ACTION Step_A_01_MoveToXY:
CASE StepA.step OF
	100:
		IF moveCmd_X < Ax_P_Limite AND moveCmd_X > Ax_N_Limite THEN
			StepA.step := StepA.step + 1;
		ELSIF moveCmd_X >= Ax_P_Limite THEN
			StepA.step := StepA.step + 10000;
			pMsg.Push_Alarm("GroupA MoveXY:命令位置超出X軸+極限");
		ELSE
			StepA.step := StepA.step + 10000;
			pMsg.Push_Alarm("GroupA MoveXY:命令位置超出X軸-極限");
		END_IF
 
			
	101:
		IF moveCmd_Y < Ay_P_Limite AND moveCmd_Y > Ay_N_Limite THEN
			StepA.step := StepA.step + 1;
		ELSIF moveCmd_Y >= Ay_P_Limite THEN
			StepA.step := StepA.step + 10000;
			pMsg.Push_Alarm("GroupA MoveXY:命令位置超出Y軸+極限");
		ELSE
			StepA.step := StepA.step + 10000;
			pMsg.Push_Alarm("GroupA MoveXY:命令位置超出Y軸-極限");
		END_IF
		
	102:
		StepA.step := 110;
		
	110:
		Ax.AbsMove(moveCmd_X, moveCmd_Spd);
		Ay.AbsMove(moveCmd_Y, moveCmd_Spd);
		StepA.step := StepA.step + 1;
		
	111:
		IF (Axs.bBuzy OR Axs.bError) AND (Ays.bBuzy OR Ays.bError) THEN
			StepA.step := StepA.step + 1;
		END_IF
		
	112:
		IF Axs.bDone AND Ays.bDone THEN
			StepA.step := StepA.step + 1;
		ELSIF Axs.bError OR Ays.bError THEN
			StepA.step := StepA.step + 10000;
		END_IF
		
	113:
		StepA.bDone := TRUE;
		StepA.step := 0;
		
END_CASE
END_ACTION

ACTION Step_A_02_FindZ:
CASE StepA.step OF
	200:
		IF ProjectData.Now_Steel.Height <= 200 OR 
			Ay.Pos > posc.pos_GbY_stanby THEN
			
			StepA.step := 210;
		ELSE
			StepA.step := 213;
		END_IF
		
		
	210:
		Ax.AbsMove(posc.pos_GbX_stanby, SpdC.HighSpeed);
		Ay.AbsMove(posc.pos_GbY_stanby, SpdC.HighSpeed);
		StepA.step := StepA.step + 1;
		
	211:
		IF (Axs.bBuzy OR Azs.bError) AND (Ays.bBuzy OR Ays.bError) THEN
			StepA.step := StepA.step + 1;
		END_IF
		
	212:
		IF Axs.bDone AND Ays.bDone THEN
			StepA.step := StepA.step + 1;
		ELSIF Axs.bError OR Ays.bError THEN
			StepA.step := StepA.step + 10000;
		END_IF
		
		
	213:
		tmpPos_Z := (ProjectData.Now_Steel.Width / 2) + MaCfg.laserB_Dis + MaCfg.laserB_Z_ReferencePos;
		Az.AbsMove(tmpPos_Z, SpdC.HighSpeed);
		StepA.step := StepA.step + 1;
		
	214:
		IF Azs.bBuzy OR Azs.bError THEN
			StepA.step := StepA.step + 1;
		END_IF
		
	215:
		IF Azs.bDone THEN
			StepA.step := StepA.step + 1;
		ELSIF DisSensor_Dis > 0 AND DisSensor_Dis < 50 THEN
			 Az.Stop();
			 StepA.step := StepA.step + 1;
		ELSIF Azs.bError THEN
			StepA.step := StepA.step + 10000;
		END_IF
		
	216:
		tmr01A.IN := TRUE;
		tmr01A.PT := T#2S;
		IF tmr01A.Q THEN
			tmr01A.IN := FALSE;
			StepA.step := StepA.step + 1;
		END_IF
		
	217:
		StepA.step := 220;
		
		
	220:
		tmpPos_X := macfg.laserB_X_DisSensor2LaserCenter + 10;
		IF ProjectData.Now_Steel.Height > 200 THEN
			tmpPos_Y := (macfg.laserB_Y_ReferencePos - ProjectData.Now_Steel.Height) + 150;
		ELSE
			tmpPos_Y := (macfg.laserB_Y_ReferencePos - MaCfg.laserB_Y_DisSensor2LaserCenter) - 50;
		END_IF
		
		StepA.step := StepA.step + 1;
		
	221:
		Ax.AbsMove(tmpPos_X, SpdC.HighSpeed);
		Ay.AbsMove(tmpPos_Y, SpdC.HighSpeed);
		StepA.step := StepA.step + 1;
		
	222:
		IF (Axs.bBuzy OR Axs.bError) AND (Ays.bBuzy OR Ays.bError) THEN
			StepA.step := StepA.step + 1;
		END_IF
		
	223:
		IF Axs.bDone AND Ays.bDone THEN
			StepA.step := StepA.step + 1;
		ELSIF Axs.bError OR Ays.bError THEN
			StepA.step := StepA.step + 10000;
		END_IF
		
	224:
		StepA.step := 230;
		
		
	230: // 再280-310之間
		IF 280 < DisSensor_Dis AND DisSensor_Dis < 310 THEN
			StepA.step := 240;
		ELSE
			StepA.step := StepA.step + 1;
		END_IF
		
	231:
		Ay.AbsMove(_Position:= PosC.GbX_P_Limite - 120, SpdC.DotSpeed);
		StepA.step := StepA.step + 1;
		
	232:
		IF (280 < DisSensor_Dis AND DisSensor_Dis < 310) OR Ays.bBuzy OR Ays.bError THEN
			StepA.step := StepA.step + 1;
		END_IF
		
	233:
		IF (280 < DisSensor_Dis AND DisSensor_Dis < 310) THEN
			Ay.Stop();
			StepA.step := StepA.step + 1;
		ELSIF Ays.bDone THEN
			pMsg.Push_Error("GroupB_FindZ:再有效距離內找不到可量測的點");
			StepA.step := StepA.step + 10000;
		ELSIF Ays.bError THEN
			StepA.step := StepA.step + 10000;
		END_IF
		
	234:
		tmr01A.IN := TRUE;
		tmr01A.PT := T#2S;
		IF tmr01A.Q THEN
			tmr01A.IN := FALSE;
			StepA.step := StepA.step + 1;
		END_IF
		
	235:
		Ay.RelMove(3, SpdC.LowSpeed);
		StepA.step := StepA.step + 1;
		
	236:
		IF Ays.bBuzy OR Ays.bError THEN
			StepA.step := StepA.step + 1;
		END_IF
		
	237:
		IF Ays.bDone THEN
			StepA.step := StepA.step + 1;
		ELSIF Ays.bError THEN
			StepA.step := StepA.step + 10000;
		END_IF
		
	238:
		StepA.step := 240;
		
		
	240:
		moveZdis := DisSensor_Dis - Macfg.laserB_Dis;
		StepA.step := StepA.step + 1;
	
	241:
		Az.RelMove(moveZdis * -1, SpdC.HighSpeed);
		StepA.step := StepA.step + 1;
		
	242:
		IF Azs.bBuzy OR Azs.bError THEN
			StepA.step := StepA.step + 1;
		END_IF
		
	243:
		IF Azs.bDone THEN
			StepA.step := StepA.step + 1;
		ELSIF Azs.bError THEN
			StepA.step := StepA.step + 10000;
		END_IF
		
	244:
		tmr01A.IN := TRUE;
		tmr01A.PT := T#2S;
		IF tmr01A.Q THEN
			tmr01A.IN := FALSE;
			StepA.step := StepA.step + 1;
		END_IF
		
	245:
		StepA.step := 250;
		
		
	250:
		moveZdis := DisSensor_Dis - Macfg.laserB_Dis;
		IF ProjectData.Now_Steel.Height > 200 THEN
			tmpPos_Y := (macfg.laserB_Y_ReferencePos - ProjectData.Now_Steel.Height) + 125;
		ELSE
			tmpPos_Y := macfg.laserB_Y_ReferencePos - (ProjectData.Now_Steel.Height / 2);
		END_IF
		StepA.step := StepA.step + 1;
		
	251:
		Az.RelMove(moveZdis * -1, SpdC.LowSpeed);
		Ay.AbsMove(tmpPos_Y, SpdC.HighSpeed);
		StepA.step := StepA.step + 1;
		
	252:
		IF (Ays.bBuzy OR Ays.bError) AND (Azs.bBuzy OR Azs.bError) THEN
			StepA.step := StepA.step + 1;
		END_IF
		
	253:
		IF Ays.bDone AND Azs.bDone THEN
			StepA.step := StepA.step + 1;
		ELSIF Azs.bError THEN
			StepA.step := StepA.step + 10000;
		END_IF
		
	254:
		StepA.step := 260;
		
	260:
		z_PosMeasure := Az.Pos;
		StepA.bDone := TRUE;
		StepA.step	:= 0;
		
END_CASE
END_ACTION

ACTION Step_A_03_FindY:
CASE StepA.step OF
	300: // 判斷當距離再200~400間，才做偵測
		IF DisSensor_Dis > 200 OR DisSensor_Dis < 400 THEN
			StepA.step := StepA.step + 1;
		ELSE
			pmsg.Push_Alarm_NoPause("GroupB:Z軸距離感應器不再感應範圍內，取消Y軸原點偵測，使用預設值");
			StepA.step	:= 380;
		END_IF
		
	301:
		StepA.step := 310;
		
	310: 
		Ay.AbsMove(100, 50);
		StepA.step := StepA.step + 1;
		
	311:
		IF Ays.bBuzy OR Ays.bError THEN
			StepA.step := StepA.step + 1;
		END_IF
		
	312:
		IF NOT DisSensor_SSC1 THEN
			Ay.Stop();
			StepA.step := StepA.step + 1;
		ELSIF Ays.bDone THEN
			pmsg.Push_Alarm_NoPause("GroupB:Z軸距離感應器訊號錯誤");
			StepA.step := 380;
		ELSIF Ays.bError THEN
			StepA.step := StepA.step + 10000;
		END_IF
		
	313:
		tmr01A.IN := TRUE;
		tmr01A.PT := T#500MS;
		IF tmr01A.Q THEN
			tmr01A.IN := FALSE;
			StepA.step := StepA.step + 1;
		END_IF
		
	314:
		StepA.step := 320;
		
	320:
		Ay.AbsMove(Ay_P_Limite - 5, 5);
		StepA.step := StepA.step + 1;
		
	321:
		IF (Ays.bBuzy OR Ays.bError) THEN
			StepA.step := StepA.step + 1;
		END_IF
		
	322:
		IF DisSensor_SSC1 THEN
			Ay.Stop();
			StepA.step := StepA.step + 1;
		ELSIF Ays.bDone THEN
			pmsg.Push_Alarm_NoPause("GroupB:Z軸距離感應器訊號錯誤");
			StepA.step := 380;
		ELSIF Ays.bError THEN
			StepA.step := StepA.step + 10000;
		END_IF
		
	323:
		tmr01A.IN := TRUE;
		tmr01A.PT := T#500MS;
		IF tmr01A.Q THEN
			tmr01A.IN := FALSE;
			StepA.step := StepA.step + 1;
		END_IF
		
	324:
		StepA.step := 330;
		
		
	330:
		Ay.AbsMove(100, 0.5);
		StepA.step := StepA.step + 1;
		
	331:
		IF Ays.bBuzy OR Ays.bError THEN
			StepA.step := StepA.step + 1;
		END_IF
		
	332:
		IF NOT DisSensor_SSC1 THEN
			Ay.Stop();
			StepA.step := StepA.step + 1;
		ELSIF Ays.bDone THEN
			pmsg.Push_Alarm_NoPause("GroupB:Z軸距離感應器訊號錯誤");
			StepA.step := 380;
		ELSIF Ays.bError THEN
			StepA.step := StepA.step + 10000;
		END_IF
		
	333:
		tmr01A.IN := TRUE;
		tmr01A.PT := T#500MS;
		IF tmr01A.Q THEN
			tmr01A.IN := FALSE;
			StepA.step := StepA.step + 1;
		END_IF
		
	334:
		StepA.step := 340;
		
		
	340:
		Set_Y_Ref(Ay.Pos);
		StepA.step := StepA.step + 1;
		
	341:
		StepA.step := 390;
		
	
	380:
		IF projectData.Now_Steel.Height > 0 THEN
			Set_Y_Ref(Ay_P_Limite + 56 - projectData.Now_Steel.Height);
		ELSE
			Set_Y_Ref(Ay_P_Limite + 56 - 500);
		END_IF
		StepA.step := StepA.step + 1;
		
	381:
		StepA.step	:= 390;
	
	390:
		StepA.bDone := TRUE;
		StepA.step	:= 0;
		
END_CASE
END_ACTION

ACTION Step_A_10_MoveToXY_REF:
CASE StepA.step OF
	1000:// 計算相對距離
		tmpPos_X := moveCmd_X - pointRef.X;
		tmpPos_Y := moveCmd_Y + pointRef.Y;
		Dxf_Y_Move := 0;
		StepA.step := StepA.step + 1;
		
	1001:
		IF tmpPos_X < Ax_P_Limite AND tmpPos_X > Ax_N_Limite THEN
			StepA.step := StepA.step + 1;
		ELSIF tmpPos_X >= Ax_P_Limite THEN
			StepA.step := StepA.step + 10000;
			pMsg.Push_Alarm("GroupB MoveXY:命令位置超出X軸+極限");
		ELSE
			StepA.step := StepA.step + 10000;
			pMsg.Push_Alarm("GroupB MoveXY:命令位置超出X軸-極限");
		END_IF
 
			
	1002:
		IF tmpPos_Y < Ay_P_Limite AND tmpPos_Y > Ay_N_Limite THEN
			StepA.step := StepA.step + 1;
		ELSIF tmpPos_Y >= Ay_P_Limite THEN
			StepA.step := StepA.step + 10000;
			pMsg.Push_Alarm("GroupB MoveXY_Ref:命令位置超出Y軸+極限");
		ELSE
			StepA.step := StepA.step + 10000;
			pMsg.Push_Alarm("GroupB MoveXY_Ref:命令位置超出Y軸-極限");
		END_IF
		
	1003:
		StepA.step := 1010;
		
	1010:
		Ax.AbsMove(tmpPos_X, moveCmd_Spd);
		Ay.AbsMove(tmpPos_Y, moveCmd_Spd);
		StepA.step := StepA.step + 1;
		
	1011:
		IF (Axs.bBuzy OR Axs.bError) AND (Ays.bBuzy OR Ays.bError) THEN
			StepA.step := StepA.step + 1;
		END_IF
		
	1012:
		IF Axs.bDone AND Ays.bDone THEN
			StepA.step := StepA.step + 1;
		ELSIF Axs.bError OR Ays.bError THEN
			StepA.step := StepA.step + 10000;
		END_IF
		
	1013:
		tmr01A.IN := TRUE;
		tmr01A.PT := T#1S;
		IF tmr01A.Q THEN
			tmr01A.IN := FALSE;
			StepA.step := StepA.step + 1;
		END_IF
		
	1014:
		StepA.step := 1020;
		
	1020:
		StepA.bDone := TRUE;
		StepA.step := 0;
		
END_CASE
END_ACTION

ACTION Step_A_20_ToStanbyPos:
CASE StepA.step OF
	2000:
		StepA.step := 2010;
		
	2010:
		IF Az.Pos > posc.pos_GbZ_stanby - 20 THEN
			StepA.step := 2020;
		ELSE
			StepA.step := StepA.step + 1;
		END_IF
		
	2011:
		Az.RelMove(20, SpdC.HomeSpeed);
		StepA.step := StepA.step + 1;
		
	2012:
		IF Azs.bDone OR Azs.bError OR NOT GbZ.outLimiter THEN
			StepA.step := StepA.step + 1;
		END_IF
		
	2013:
		IF Azs.bDone OR NOT GbZ.outLimiter THEN
			StepA.step := StepA.step + 1;
		ELSIF Azs.bError THEN
			StepA.step := StepA.step + 10000;
		END_IF
		
	2014:
		StepA.step := 2020;
		
	2020:
		Ax.AbsMove(posc.pos_GbX_stanby, moveCmd_Spd);
		StepA.step := StepA.step + 1;
		
	2021:
		IF (Axs.bBuzy OR Axs.bError) THEN
			StepA.step := StepA.step + 1;
		END_IF
		
	2022:
		IF Axs.bDone THEN
			StepA.step := StepA.step + 1;
		ELSIF Axs.bError THEN
			StepA.step := StepA.step + 10000;
		END_IF
	
	2023:
		StepA.step := 2030;
	
	2030:
		Az.AbsMove(posc.pos_GbZ_stanby, moveCmd_Spd);
		Ay.AbsMove(posc.pos_GbY_stanby, moveCmd_Spd);
		StepA.step := StepA.step + 1;
		
	2031:
		IF (Azs.bBuzy OR Azs.bError) AND (Ays.bBuzy OR Ays.bError)  THEN
			StepA.step := StepA.step + 1;
		END_IF
		
	2032:
		IF Azs.bDone AND Ays.bDone THEN
			StepA.step := StepA.step + 1;
		ELSIF Azs.bError OR Ays.bError THEN
			StepA.step := StepA.step + 10000;
		END_IF
		
	2033:
		StepA.step := 2040;
		
		
	2040:
		StepA.bDone := TRUE;
		StepA.step := 0;
		
END_CASE
END_ACTION

ACTION Timer:
tmr01A();
tmr01();
tmr02();

// tmr_oil(in := IO.q205 AND IO.i402, PT:=T#2S);
tmr_oil(in := IO.q205, PT:=T#2S);

IF tmr_oil.Q THEN
	IO.q205 := FALSE;
	
	Axis.GbX_Last_Oil := Axis.GbX_total_Move;
	
	Axis.GbY_Last_Oil := Axis.GbY_total_Move;
	
	Axis.GbZ_Last_Oil := Axis.GbZ_total_Move;
END_IF
END_ACTION

METHOD ToStanby : BOOL
VAR_INPUT
	Speed : LREAL := 0;
END_VAR
StepA.bDone := FALSE;
IF Speed > 0 THEN
	moveCmd_Spd := Speed;
ELSE
	moveCmd_Spd := SpdC.HomeSpeed;
END_IF

// ============ 紀錄啟動條件 ============
_logA.fbJson.StartObject();
_logA.fbJson.AddKeyString('MethodName','ToStanby');
_logA.fbJson.AddKeyLreal('Velocity', Speed);
_logA.JsonOutput();
// ======================================



StepA.step := 2000;
END_METHOD

METHOD XY_Move : BOOL
VAR_INPUT
	X_Point : REAL;
	Y_Point	: REAL;
	Speed : REAL;
END_VAR
moveCmd_X := X_Point;
moveCmd_Y := Y_Point;
moveCmd_Spd := Speed;

StepA.bDone := FALSE;

// ============ 紀錄啟動條件 ============
_logA.fbJson.StartObject();
_logA.fbJson.AddKeyString('MethodName','XY_Move');
_logA.fbJson.AddKeyLreal('X_Point', X_Point);
_logA.fbJson.AddKeyLreal('Y_Point', Y_Point);
_logA.fbJson.AddKeyLreal('Velocity', Speed);
_logA.JsonOutput();
// ======================================



StepA.step := 100;
END_METHOD

METHOD XY_Move_Ref : BOOL
VAR_INPUT
	X_Point : LREAL;
	Y_Point	: LREAL;
	Speed : LREAL;
END_VAR
moveCmd_X := X_Point;
moveCmd_Y := Y_Point;
moveCmd_Spd := Speed;

StepA.bDone := FALSE;

// ============ 紀錄啟動條件 ============
_logA.fbJson.StartObject();
_logA.fbJson.AddKeyString('MethodName','XY_Move_Ref');
_logA.fbJson.AddKeyLreal('X_Point', X_Point);
_logA.fbJson.AddKeyLreal('Y_Point', Y_Point);
_logA.fbJson.AddKeyLreal('Velocity', Speed);
_logA.JsonOutput();
// ======================================



StepA.step := 1000;
END_METHOD

END_PROGRAM

// ---- POUs/動作流程控制/AxisGroup功能塊/GroupC.TcPOU
PROGRAM GroupC
VAR
	step		: INT;
	
	StepA		: Sub_Step;
	
	// X軸映射
	Ax : I_Axis;
	Axs: Sub_Step;
	// Y軸映射
	Ay : I_Axis;
	Ays: Sub_Step;
	// X軸映射
	Az : I_Axis;
	Azs: Sub_Step;
	
	Ax_P_Limite : LREAL;
	Ax_N_Limite : LREAL;
	Ay_P_Limite : LREAL;
	Ay_N_Limite : LREAL;
	Az_P_Limite : LREAL;
	Az_N_Limite : LREAL;

	
	// 移動命令的 X位置
	moveCmd_X: LREAL;
	// 移動命令的 Y位置
	moveCmd_Y: LREAL;
	// 移動命令 速度
	moveCmd_Spd: LREAL;
	
	moveZdis	: REAL;
	tmr01A		: TON;
	tmr01		: TON;
	tmr02		: TON;
	
	// 坐標系的參考原點
	pointRef : XYZ_Point;
	
	// 移動位置X 計算結果
	tmpPos_X: LREAL;
	// 移動位置Y 計算結果
	tmpPos_Y: LREAL;
	// 移動位置Z 計算結果
	tmpPos_Z: LREAL;
	
	// 雷射圖形移動距離 Y
	Dxf_Y_Move : LREAL;
	

	// 測量到的Z位置
	z_PosMeasure: REAL;
	
	// 距離感應器IO
	DisSensor_SSC1: BOOL;
	// 距離感應器距離
	DisSensor_Dis: LREAL;
	
	Boot : BOOL := TRUE;
	
	
	
	// 執行中的清單號
	WorkNum: INT;
	
	// 鏡頭 吹氣
	q_Lens_Blow :BOOL;
	
	// 重試計數器
	_retryCnt: INT;
	
	// 可以開始雕刻 (Fx就緒)
	_ReadyToPrint :BOOL;
	// 可以開始移動 (Fx就緒)
	_ReadyToMove :BOOL;
	
	
	// 計算上次打油後的一棟距離
	X_Move: LREAL;
	Y_Move: LREAL;
	Z_Move: LREAL;
	tmr_oil: TON;
	
	_log : Step_Log; 
	_logA : Step_Log; 
	sql_hand: UDINT;
END_VAR



VAR_OUTPUT
	// 工件高度
	Size_H : REAL;
	// 工件座標
	RefPos : XYZ_Point;
	
	// 功能執行中
	bBuzy 	: BOOL;
	// 功能結束
	bDone	: BOOL;
	// 發生錯誤
	bError	: BOOL;
END_VAR

IF Boot THEN
	Ax := axis.GcX;
	Ay := axis.GcY;
	Az := axis.GcZ;
	boot := FALSE;
END_IF

Axs := Ax.State;
Ays := Ay.State;
Azs := Az.State;

Ax_P_Limite := posc.GcX_P_Limite;
Ax_N_Limite := posc.GcX_N_Limite;
Ay_P_Limite := posc.GcY_P_Limite;
Ay_N_Limite := posc.GcY_N_Limite;
Az_P_Limite := posc.GcZ_P_Limite;
Az_N_Limite := posc.GcZ_N_Limite;

DisSensor_SSC1	:= Sensor.sensorC.SSC1_1;
DisSensor_Dis	:= Sensor.sensorC.Distance;

IF (EStop OR SystemError) THEN
	IF bBuzy THEN
		step := step  + 10000;
	END_IF
	IF StepA.bBuzy THEN
		StepA.step := StepA.step  + 10000;
	END_IF
	Hmi_Web.Process_Data_UUID_C_Start := FALSE;
	q_Lens_Blow := FALSE;
END_IF

bBuzy := step > 0 AND step < 10000;
bError := step >= 10000;
IF bBuzy OR bError THEN
	bDone := FALSE;
END_IF

Step_01_DoPayloadList();
Step_02_Do_2nd_in_list();
Step_03_DoLaserAction();



StepA.bBuzy := StepA.step > 0 AND StepA.step < 10000;
StepA.bError := StepA.step >= 10000;
IF StepA.bBuzy OR StepA.bError THEN
	StepA.bDone := FALSE;
END_IF

Step_A_01_MoveToXY();
Step_A_02_FindZ();
Step_A_03_FindY();
Step_A_10_MoveToXY_REF();
Step_A_20_ToStanbyPos();

Timer();

RefPos.X := Ax.Pos - pointRef.X;
RefPos.Y := Ay.Pos - pointRef.Y;
RefPos.Z := Az.Pos - pointRef.Z;

ProjectData.Now_Steel_Payload_C_DataNumberDone := WorkNum;

io.q307 := q_Lens_Blow;

_log(name:= 'GroupC', step:= step);
_logA(name:= 'GroupC_Mov', step:= StepA.Step);

METHOD Do_WorkList : BOOL
VAR_INPUT
END_VAR
bDone := FALSE;

// ============ 紀錄啟動條件 ============
_log.fbJson.StartObject();
_log.fbJson.AddKeyString('MethodName','Do_WorkList');
_log.JsonOutput();
// ======================================




Step := 100;
END_METHOD

METHOD FindZ : BOOL
VAR_INPUT
END_VAR
StepA.bDone := FALSE;

// ============ 紀錄啟動條件 ============
_logA.fbJson.StartObject();
_logA.fbJson.AddKeyString('MethodName','FindZ');
_logA.JsonOutput();
// ======================================






StepA.step := 200;
END_METHOD

METHOD FindZ_Fast : BOOL
VAR_INPUT
END_VAR
StepA.bDone := FALSE;

// ============ 紀錄啟動條件 ============
_logA.fbJson.StartObject();
_logA.fbJson.AddKeyString('MethodName','FindZ_Fast');
_logA.JsonOutput();
// ======================================





StepA.step := 220;
END_METHOD

ACTION Oil:
X_Move := Axis.GcX_total_Move - Axis.GcX_Last_Oil;
Y_Move := Axis.GcY_total_Move - Axis.GcY_Last_Oil;
Z_Move := Axis.GcZ_total_Move - Axis.GcZ_Last_Oil;

IF X_Move > 1000000 OR Y_Move > 1000000 OR Z_Move > 1000000 THEN
	IO.q206 := TRUE;
END_IF
END_ACTION

PROPERTY ReadyToMove : BOOL
GET
ReadyToMove := _ReadyToMove;
END_GET
SET
_ReadyToMove := ReadyToMove;
END_SET
END_PROPERTY

PROPERTY ReadyToPrint : BOOL
GET
ReadyToPrint := _ReadyToPrint;
END_GET
SET
_ReadyToPrint := ReadyToPrint;
END_SET
END_PROPERTY

METHOD Set_X_Ref
VAR_INPUT
	Value : LREAL;
END_VAR
pointRef.X := Value;
END_METHOD

METHOD Set_Y_Ref
VAR_INPUT
	Value : LREAL;
END_VAR
pointRef.Y := Value;
END_METHOD

ACTION Step_01_DoPayloadList:
CASE step OF
(*	===============================================
		開始做 Payload_B_Data_buff 清單內的工作
	===============================================*)
	100: // 以數量判斷是否有工作
		WorkNum := 0;
		IF ProjectData.Now_Steel_Payload_C_DataNumber > 0 THEN
			step := step + 1;
		ELSE
			bDone := TRUE;
			Step := 0;
		END_IF
 
			
	101:
		// 初始化工作暫存器
		Hmi_Web.Process_Data_UUID_A_Start := FALSE;
		WorkNum := 0;
		step := 110;
		
(*	===============================================
					設定工作中的專案
	===============================================*)
	110:
		ProjectData.Payload_C_Data_Now := ProjectData.Payload_C_Data_buff[WorkNum];
		Hmi_Web.Process_Data_UUID_A := ProjectData.Payload_C_Data_buff[WorkNum].data_uid;
		step := step + 1;
	
	111:
		step := 120;
		
(*	===============================================
					移動到位置
	===============================================*)
	120:
		IF _ReadyToMove THEN
			step := step + 1;
		END_IF
		
	121:
		XY_Move_Ref(
			ProjectData.Payload_C_Data_Now.Point_X, 
			ProjectData.Payload_C_Data_Now.Point_Y, 
			SpdC.HighSpeed
		);
		step := step + 1;
		
	122:
		IF stepA.bBuzy OR stepA.bError THEN
			step := step + 1;
		END_IF
		
	123:
		IF stepA.bDone THEN
			step := step + 1;
		ELSIF stepA.bError THEN
			step := step + 10000;
		END_IF
		
	124:
		step := 130;
	

(*	===============================================
				雷射主機 啟動 預覽/雕刻 動作
	===============================================*)	
	130:
		step := 300;
END_CASE
END_ACTION

ACTION Step_02_Do_2nd_in_list:
CASE step OF
	200:
		step := 210;
		
(*	===============================================
					設定工作中的專案
	===============================================*)
	210:
		ProjectData.Payload_C_Data_Now := ProjectData.Payload_C_Data_buff[WorkNum];
		Hmi_Web.Process_Data_UUID_A := ProjectData.Payload_C_Data_buff[WorkNum].data_uid;
		step := step + 1;
	
	211:
		step := 220;
		
(*	===============================================
					移動到位置
	===============================================*)
	220:
		XY_Move_Ref(
			ProjectData.Payload_C_Data_Now.Point_X, 
			ProjectData.Payload_C_Data_Now.Point_Y, 
			SpdC.HighSpeed
		);
		step := step + 1;
		
	221:
		IF stepA.bBuzy OR stepA.bError THEN
			step := step + 1;
		END_IF
		
	222:
		IF stepA.bDone THEN
			step := step + 1;
		ELSIF stepA.bError THEN
			step := step + 10000;
		END_IF
		
	223:
		step := 230;

(*	===============================================
				雷射主機 啟動 預覽/雕刻 動作
	===============================================*)	
	230:
		step := 300;
		
END_CASE
END_ACTION

ACTION Step_03_DoLaserAction:
CASE step OF
	300:
		IF ReadyToPrint THEN
			step := step + 1;
		END_IF
		
	301:
		sql_hand := ReadSQLData.Set_Payload_Start(ProjectData.Payload_C_Data_Now.data_uid);
		IF sql_hand <> 0 THEN
			step := step + 1;
		END_IF
		
	302:
		step := 310;

(*	===============================================
				雷射主機 啟動 預覽/雕刻 動作
	===============================================*)	
	310:
		q_Lens_Blow := TRUE;
		IF LEN(Hmi_Web.Process_Data_UUID_A) = 0 THEN
			Hmi_Web.Process_Data_UUID_A := ProjectData.Payload_C_Data_buff[WorkNum].data_uid;
		ELSE
			step := step + 1;
		END_IF
		
	311:
		Hmi_Web.Process_Data_UUID_A_Start := TRUE;
		// ============ 紀錄啟動條件 ============
		_log.fbJson.StartObject();
		_log.fbJson.AddKeyString('StepName','Laser_C_Start');
		_log.fbJson.AddKeyBool('Process_Data_UUID_A_Start', Hmi_Web.Process_Data_UUID_A_Start);
		_log.fbJson.AddKeyString('Payload_C_Data_Now', ProjectData.Payload_C_Data_Now.data_uid);
		_log.JsonOutput();
		// ======================================
		step := step + 1;
		
	312:	
		tmr01.PT := T#500MS;
		tmr01.IN := TRUE;
		IF tmr01.Q THEN
			tmr01.IN := FALSE;
			tmr02.IN := FALSE;
			step := step + 1;
		END_IF
		
	313:
		tmr01.PT := TO_TIME(MaCfg.LaserPrinter_Timeout);
		tmr01.IN := TRUE;
		tmr02.PT := T#250mS;
		tmr02.IN := NOT Hmi_Web.Process_Data_UUID_A_Start;
		IF tmr02.Q THEN
			Hmi_Web.Process_Data_UUID_A :='';
			tmr01.IN := FALSE;
			tmr02.IN := FALSE;
			// ============ 紀錄啟動條件 ============
			_log.fbJson.StartObject();
			_log.fbJson.AddKeyString('StepName','Laser_C_Done');
			_log.JsonOutput();
			// ======================================
			step := step + 1;
		ELSIF tmr01.Q THEN
			tmr01.IN := FALSE;
			tmr02.IN := FALSE;
			pMsg.Push_Error("GroupC:雷射動作超時");
			step := step + 10000;
		END_IF
	
	314:
		WorkNum := WorkNum + 1;
		q_Lens_Blow := FALSE;
		step := 320;
		
(*	================================================
				開始下個循環或此區域結束
	================================================*)	
	320:
		sql_hand := ReadSQLData.Set_Payload_Finish(ProjectData.Payload_C_Data_Now.data_uid);
		IF sql_hand <> 0 THEN
			step := step + 1;
		END_IF
	
	321:
		IF WorkNum < ProjectData.Now_Steel_Payload_C_DataNumber THEN
		// 這個區域還有工作
			step := step + 1;
		ELSE
		// 這個區域工作結束
			step := 390;
		END_IF
		
	322:
		// 設定工作中的專案
		step := 200;
		
(*	================================================
				此區域結束
	================================================*)		
	390:
		bDone := TRUE;
		step := 0;
END_CASE
END_ACTION

ACTION Step_A_01_MoveToXY:
CASE StepA.step OF
	100:
		IF moveCmd_X < Ax_P_Limite AND moveCmd_X > Ax_N_Limite THEN
			StepA.step := StepA.step + 1;
		ELSIF moveCmd_X >= Ax_P_Limite THEN
			StepA.step := StepA.step + 10000;
			pMsg.Push_Alarm("GroupA MoveXY:命令位置超出X軸+極限");
		ELSE
			StepA.step := StepA.step + 10000;
			pMsg.Push_Alarm("GroupA MoveXY:命令位置超出X軸-極限");
		END_IF
 
			
	101:
		IF moveCmd_Y < Ay_P_Limite AND moveCmd_Y > Ay_N_Limite THEN
			StepA.step := StepA.step + 1;
		ELSIF moveCmd_Y >= Ay_P_Limite THEN
			StepA.step := StepA.step + 10000;
			pMsg.Push_Alarm("GroupA MoveXY:命令位置超出Y軸+極限");
		ELSE
			StepA.step := StepA.step + 10000;
			pMsg.Push_Alarm("GroupA MoveXY:命令位置超出Y軸-極限");
		END_IF
		
	102:
		StepA.step := 110;
		
	110:
		Ax.AbsMove(moveCmd_X, moveCmd_Spd);
		Ay.AbsMove(moveCmd_Y, moveCmd_Spd);
		StepA.step := StepA.step + 1;
		
	111:
		IF (Axs.bBuzy OR Axs.bError) AND (Ays.bBuzy OR Ays.bError) THEN
			StepA.step := StepA.step + 1;
		END_IF
		
	112:
		IF Axs.bDone AND Ays.bDone THEN
			StepA.step := StepA.step + 1;
		ELSIF Axs.bError OR Ays.bError THEN
			StepA.step := StepA.step + 10000;
		END_IF
		
	113:
		StepA.bDone := TRUE;
		StepA.step := 0;
		
END_CASE
END_ACTION

ACTION Step_A_02_FindZ:
CASE StepA.step OF
	200:
		StepA.step := 220;
		
	220:
		tmpPos_X := 150;
		tmpPos_Y := (ProjectData.Now_Steel.Width / 2) + pointRef.Y;
		tmpPos_Z := ProjectData.Now_Steel.Height + MaCfg.laserC_Dis + MaCfg.laserC_Z_ReferencePos;
		StepA.step := StepA.step + 1;
		
	221:
		Ax.AbsMove(tmpPos_X, SpdC.HighSpeed);
		Ay.AbsMove(tmpPos_Y, SpdC.HighSpeed);
		Az.AbsMove(tmpPos_Z, SpdC.HighSpeed);
		StepA.step := StepA.step + 1;
		
	222:
		IF (Axs.bBuzy OR Axs.bError) AND 
			(Ays.bBuzy OR Ays.bError) AND
			(Azs.bBuzy OR Azs.bError) THEN
			StepA.step := StepA.step + 1;
		END_IF
		
	223:
		IF Axs.bDone AND Ays.bDone AND Azs.bDone THEN
			StepA.step := StepA.step + 1;
		ELSIF Axs.bError OR Ays.bError OR Azs.bError THEN
			StepA.step := StepA.step + 10000;
		END_IF
		
	224:
		StepA.step := 230;
		
	
	230: // 再280-310之間
		IF 280 < DisSensor_Dis AND DisSensor_Dis < 310 THEN
			StepA.step := 240;
		ELSE
			StepA.step := StepA.step + 1;
		END_IF
		
	231:
		Ay.AbsMove((ProjectData.Now_Steel.Width - 10) + pointRef.Y, SpdC.DotSpeed);
		StepA.step := StepA.step + 1;
		
	232:
		IF (280 < DisSensor_Dis AND DisSensor_Dis < 310) OR Ays.bBuzy OR Ays.bError THEN
			StepA.step := StepA.step + 1;
		END_IF
		
	233:
		IF (280 < DisSensor_Dis AND DisSensor_Dis < 310) THEN
			Ay.Stop();
			StepA.step := StepA.step + 1;
		ELSIF Ays.bDone THEN
			pMsg.Push_Error("GroupC_FindZ:再有效距離內找不到可量測的點");
			StepA.step := StepA.step + 10000;
		ELSIF Ays.bError THEN
			StepA.step := StepA.step + 10000;
		END_IF
		
	234:
		tmr01A.IN := TRUE;
		tmr01A.PT := T#2S;
		IF tmr01A.Q THEN
			tmr01A.IN := FALSE;
			StepA.step := StepA.step + 1;
		END_IF
		
	235:
		Ay.RelMove(3, SpdC.LowSpeed);
		StepA.step := StepA.step + 1;
		
	236:
		IF Ays.bBuzy OR Ays.bError THEN
			StepA.step := StepA.step + 1;
		END_IF
		
	237:
		IF Ays.bDone THEN
			StepA.step := StepA.step + 1;
		ELSIF Ays.bError THEN
			StepA.step := StepA.step + 10000;
		END_IF
		
	238:
		StepA.step := 240;
	
		
	240:
		moveZdis := DisSensor_Dis - Macfg.laserC_Dis;
		StepA.step := StepA.step + 1;
		
		
	241:
		Az.RelMove(moveZdis * -1, SpdC.HighSpeed);
		StepA.step := StepA.step + 1;
		
	242:
		IF Azs.bBuzy OR Azs.bError THEN
			StepA.step := StepA.step + 1;
		END_IF
		
	243:
		IF Azs.bDone THEN
			StepA.step := StepA.step + 1;
		ELSIF Azs.bError THEN
			StepA.step := StepA.step + 10000;
		END_IF
		
	244:
		tmr01A.IN := TRUE;
		tmr01A.PT := T#2S;
		IF tmr01A.Q THEN
			tmr01A.IN := FALSE;
			StepA.step := StepA.step + 1;
		END_IF
		
	245:
		StepA.step := 250;
		
		
	250:
		moveZdis := DisSensor_Dis - Macfg.laserC_Dis;
		StepA.step := StepA.step + 1;
		
	251:
		Az.RelMove(moveZdis * -1, SpdC.LowSpeed);
		StepA.step := StepA.step + 1;
		
	252:
		IF Azs.bBuzy OR Azs.bError THEN
			StepA.step := StepA.step + 1;
		END_IF
		
	253:
		IF Azs.bDone THEN
			StepA.step := StepA.step + 1;
		ELSIF Azs.bError THEN
			StepA.step := StepA.step + 10000;
		END_IF
		
	254:
		StepA.step := 260;
		
	260:
		z_PosMeasure := Az.Pos;
		StepA.bDone := TRUE;
		StepA.step	:= 0;
		
END_CASE
END_ACTION

ACTION Step_A_03_FindY:
CASE StepA.step OF
	300: // 判斷當距離再200~400間，才做偵測
		IF DisSensor_Dis > 200 OR DisSensor_Dis < 400 THEN
			StepA.step := StepA.step + 1;
		ELSE
			pmsg.Push_Alarm_NoPause("GroupC:Z軸距離感應器不再感應範圍內，取消Y軸原點偵測，使用預設值");
			StepA.step	:= 380;
		END_IF
		
	301:
		StepA.step := 310;
		
	310: 
		Ay.AbsMove(100, 50);
		StepA.step := StepA.step + 1;
		
	311:
		IF Ays.bBuzy OR Ays.bError THEN
			StepA.step := StepA.step + 1;
		END_IF
		
	312:
		IF NOT DisSensor_SSC1 THEN
			Ay.Stop();
			StepA.step := StepA.step + 1;
		ELSIF Ays.bDone THEN
			pmsg.Push_Alarm_NoPause("GroupC:Z軸距離感應器訊號錯誤");
			StepA.step := 380;
		ELSIF Ays.bError THEN
			StepA.step := StepA.step + 10000;
		END_IF
		
	313:
		tmr01A.IN := TRUE;
		tmr01A.PT := T#500MS;
		IF tmr01A.Q THEN
			tmr01A.IN := FALSE;
			StepA.step := StepA.step + 1;
		END_IF
		
	314:
		StepA.step := 320;
		
	320:
		Ay.AbsMove(Ay_P_Limite - 5, 5);
		StepA.step := StepA.step + 1;
		
	321:
		IF (Ays.bBuzy OR Ays.bError) THEN
			StepA.step := StepA.step + 1;
		END_IF
		
	322:
		IF DisSensor_SSC1 THEN
			Ay.Stop();
			StepA.step := StepA.step + 1;
		ELSIF Ays.bDone THEN
			pmsg.Push_Alarm_NoPause("GroupC:Z軸距離感應器訊號錯誤");
			StepA.step := 380;
		ELSIF Ays.bError THEN
			StepA.step := StepA.step + 10000;
		END_IF
		
	323:
		tmr01A.IN := TRUE;
		tmr01A.PT := T#500MS;
		IF tmr01A.Q THEN
			tmr01A.IN := FALSE;
			StepA.step := StepA.step + 1;
		END_IF
		
	324:
		StepA.step := 330;
		
		
	330:
		Ay.AbsMove(100, 0.5);
		StepA.step := StepA.step + 1;
		
	331:
		IF Ays.bBuzy OR Ays.bError THEN
			StepA.step := StepA.step + 1;
		END_IF
		
	332:
		IF NOT DisSensor_SSC1 THEN
			Ay.Stop();
			StepA.step := StepA.step + 1;
		ELSIF Ays.bDone THEN
			pmsg.Push_Alarm_NoPause("GroupC:Z軸距離感應器訊號錯誤");
			StepA.step := 380;
		ELSIF Ays.bError THEN
			StepA.step := StepA.step + 10000;
		END_IF
		
	333:
		tmr01A.IN := TRUE;
		tmr01A.PT := T#500MS;
		IF tmr01A.Q THEN
			tmr01A.IN := FALSE;
			StepA.step := StepA.step + 1;
		END_IF
		
	334:
		StepA.step := 340;
		
		
	340:
		Set_Y_Ref(Ay.Pos);
		StepA.step := StepA.step + 1;
		
	341:
		StepA.step := 390;
		
	
	380:
		IF projectData.Now_Steel.Width > 0 THEN
			Set_Y_Ref(Ay_P_Limite + 56 - projectData.Now_Steel.Width);
		ELSE
			Set_Y_Ref(Ay_P_Limite + 56 - 500);
		END_IF
		StepA.step := StepA.step + 1;
		
	381:
		StepA.step	:= 390;
	
	390:
		z_PosMeasure := GaZ.Pos;
		StepA.bDone := TRUE;
		StepA.step	:= 0;
		
END_CASE
END_ACTION

ACTION Step_A_10_MoveToXY_REF:
CASE StepA.step OF
	1000:// 計算相對距離
		tmpPos_X := moveCmd_X - pointRef.X;
		tmpPos_Y := moveCmd_Y + pointRef.Y;
		Dxf_Y_Move := 0;
		StepA.step := StepA.step + 1;
		
	1001:
		IF tmpPos_X < Ax_P_Limite AND tmpPos_X > Ax_N_Limite THEN
			StepA.step := StepA.step + 1;
		ELSIF tmpPos_X >= Ax_P_Limite THEN
			StepA.step := StepA.step + 10000;
			pMsg.Push_Alarm("GroupC MoveXY:命令位置超出X軸+極限");
		ELSE
			StepA.step := StepA.step + 10000;
			pMsg.Push_Alarm("GroupC MoveXY:命令位置超出X軸-極限");
		END_IF
 
			
	1002:
		IF tmpPos_Y < Ay_P_Limite AND tmpPos_Y > Ay_N_Limite THEN
			StepA.step := StepA.step + 1;
		ELSIF tmpPos_Y >= Ay_P_Limite THEN
			StepA.step := StepA.step + 10000;
			pMsg.Push_Alarm("GroupC MoveXY_Ref:命令位置超出Y軸+極限");
		ELSE
			Dxf_Y_Move := 5 - tmpPos_Y;
			Dxf_Y_Move := Dxf_Y_Move * -1;	// 雷射Y軸相反
			IF Dxf_Y_Move <= -70 THEN 
				StepA.step := StepA.step + 10000;
				pMsg.Push_Alarm("GroupC MoveXY_Ref:命令位置超出Y軸-極限");
			ELSE
				tmpPos_Y := 5;
			END_IF
		END_IF
		
	1003:
		StepA.step := 1010;
		
	1010:
		Ax.AbsMove(tmpPos_X, moveCmd_Spd);
		Ay.AbsMove(tmpPos_Y, moveCmd_Spd);
		StepA.step := StepA.step + 1;
		
	1011:
		IF (Axs.bBuzy OR Axs.bError) AND (Ays.bBuzy OR Ays.bError) THEN
			StepA.step := StepA.step + 1;
		END_IF
		
	1012:
		IF Axs.bDone AND Ays.bDone THEN
			StepA.step := StepA.step + 1;
		ELSIF Axs.bError OR Ays.bError THEN
			StepA.step := StepA.step + 10000;
		END_IF
		
	1013:
		tmr01A.IN := TRUE;
		tmr01A.PT := T#1S;
		IF tmr01A.Q THEN
			tmr01A.IN := FALSE;
			StepA.step := StepA.step + 1;
		END_IF
		
	1014:
		StepA.step := 1020;
		
	1020:
		StepA.bDone := TRUE;
		StepA.step := 0;
		
END_CASE
END_ACTION

ACTION Step_A_20_ToStanbyPos:
CASE StepA.step OF
	2000:
		StepA.step := 2030;
	
	2030:
		Ax.AbsMove(posc.pos_GcX_stanby, moveCmd_Spd);
		Ay.AbsMove(posc.pos_GcY_stanby, moveCmd_Spd);
		Az.AbsMove(posc.pos_GcZ_stanby, moveCmd_Spd);
		StepA.step := StepA.step + 1;
		
	2031:
		IF (Axs.bBuzy OR Axs.bError) AND (Ays.bBuzy OR Ays.bError) AND (Azs.bBuzy OR Azs.bError) THEN
			StepA.step := StepA.step + 1;
		END_IF
		
	2032:
		IF Axs.bDone AND Ays.bDone AND Azs.bDone THEN
			StepA.step := StepA.step + 1;
		ELSIF Axs.bError OR Ays.bError OR Azs.bError THEN
			StepA.step := StepA.step + 10000;
		END_IF
		
	2033:
		StepA.step := 2040;
		
		
	2040:
		StepA.bDone := TRUE;
		StepA.step := 0;
		
END_CASE
END_ACTION

ACTION Timer:
tmr01A();
tmr01();
tmr02();

// tmr_oil(in := IO.q206 AND IO.i410, PT:=T#2S);
tmr_oil(in := IO.q206, PT:=T#2S);

IF tmr_oil.Q THEN
	IO.q206 := FALSE;
	
	Axis.GcX_Last_Oil := Axis.GcX_total_Move;
	
	Axis.GcY_Last_Oil := Axis.GcY_total_Move;
	
	Axis.GcZ_Last_Oil := Axis.GcZ_total_Move;
END_IF
END_ACTION

METHOD ToStanby : BOOL
VAR_INPUT
	Speed : LREAL := 0;
END_VAR
StepA.bDone := FALSE;
IF Speed > 0 THEN
	moveCmd_Spd := Speed;
ELSE
	moveCmd_Spd := SpdC.HomeSpeed;
END_IF

// ============ 紀錄啟動條件 ============
_logA.fbJson.StartObject();
_logA.fbJson.AddKeyString('MethodName','ToStanby');
_logA.fbJson.AddKeyLreal('Velocity', Speed);
_logA.JsonOutput();
// ======================================




StepA.step := 2000;
END_METHOD

METHOD XY_Move : BOOL
VAR_INPUT
	X_Point : LREAL;
	Y_Point	: LREAL;
	Speed : LREAL;
END_VAR
moveCmd_X := X_Point;
moveCmd_Y := Y_Point;
moveCmd_Spd := Speed;

StepA.bDone := FALSE;

// ============ 紀錄啟動條件 ============
_logA.fbJson.StartObject();
_logA.fbJson.AddKeyString('MethodName','XY_Move');
_logA.fbJson.AddKeyLreal('X_Point', X_Point);
_logA.fbJson.AddKeyLreal('Y_Point', Y_Point);
_logA.fbJson.AddKeyLreal('Velocity', Speed);
_logA.JsonOutput();
// ======================================



StepA.step := 100;
END_METHOD

METHOD XY_Move_Ref : BOOL
VAR_INPUT
	X_Point : LREAL;
	Y_Point	: LREAL;
	Speed : LREAL;
END_VAR
moveCmd_X := X_Point;
moveCmd_Y := Y_Point;
moveCmd_Spd := Speed;

StepA.bDone := FALSE;

// ============ 紀錄啟動條件 ============
_logA.fbJson.StartObject();
_logA.fbJson.AddKeyString('MethodName','XY_Move_Ref');
_logA.fbJson.AddKeyLreal('X_Point', X_Point);
_logA.fbJson.AddKeyLreal('Y_Point', Y_Point);
_logA.fbJson.AddKeyLreal('Velocity', Speed);
_logA.JsonOutput();
// ======================================



StepA.step := 1000;
END_METHOD

END_PROGRAM

// ---- POUs/動作流程控制/AxisGroup功能塊/GroupD.TcPOU
PROGRAM GroupD
VAR
	step		: INT;
	
	StepA		: Sub_Step;
	
	// X軸映射
	Ax : I_Axis;
	Axs: Sub_Step;
	// Y軸映射
	Ay : I_Axis;
	Ays: Sub_Step;
	// X軸映射
	Az : I_Axis;
	Azs: Sub_Step;
	
	Ax_P_Limite : LREAL;
	Ax_N_Limite : LREAL;
	Ay_P_Limite : LREAL;
	Ay_N_Limite : LREAL;
	Az_P_Limite : LREAL;
	Az_N_Limite : LREAL;
	
	// 移動命令的 X位置
	moveCmd_X: LREAL;
	// 移動命令的 Y位置
	moveCmd_Y: LREAL;
	// 移動命令 速度
	moveCmd_Spd: LREAL;
	
	moveZdis	: REAL;
	tmr01A		: TON;
	tmr01		: TON;
	tmr02		: TON;
	
	// 坐標系的參考原點
	pointRef : XYZ_Point;
	
	// 移動位置X 計算結果
	tmpPos_X: LREAL;
	// 移動位置Y 計算結果
	tmpPos_Y: LREAL;
	// 移動位置Z 計算結果
	tmpPos_Z: LREAL;
	
	// 雷射圖形移動距離 Y
	Dxf_Y_Move : LREAL;
	

	// 測量到的Z位置
	z_PosMeasure: REAL;
	
	// 距離感應器IO
	DisSensor_SSC1: BOOL;
	// 距離感應器距離
	DisSensor_Dis: LREAL;
	
	Boot : BOOL := TRUE;
	
	
	
	// 執行中的清單號
	WorkNum: INT;
	
	

	// 鏡頭蓋 開 輸出
	i_Lens_Cap_IsOpen :BOOL;
	// 鏡頭蓋 關 輸出
	i_Lens_Cap_IsClose :BOOL;
	
	
	// 鏡頭蓋 開 輸出
	q_Lens_Cap_Open :BOOL;
	// 鏡頭蓋 關 輸出
	q_Lens_Cap_Close :BOOL;
	
	// 鏡頭 吹氣
	q_Lens_Blow :BOOL;
	
	
	_retryCnt: INT;
	
	// 可以開始雕刻 (Fx就緒)
	_ReadyToPrint :BOOL;
	// 可以開始移動 (Fx就緒)
	_ReadyToMove :BOOL;
	
	
	// 計算上次打油後的一棟距離
	X_Move: LREAL;
	Y_Move: LREAL;
	Z_Move: LREAL;
	tmr_oil: TON;
	
	_log : Step_Log; 
	_logA : Step_Log; 
	sql_hand: UDINT;
	tmpPos_Y1: LREAL;
END_VAR


VAR_OUTPUT
	// 工件高度
	Size_H : REAL;
	// 工件座標
	RefPos : XYZ_Point;
	
	// 功能執行中
	bBuzy 	: BOOL;
	// 功能結束
	bDone	: BOOL;
	// 發生錯誤
	bError	: BOOL;
END_VAR

IF Boot THEN
	Ax := axis.GdX;
	Ay := axis.GdY;
	Az := axis.GdZ;
	boot := FALSE;
END_IF

Axs := Ax.State;
Ays := Ay.State;
Azs := Az.State;

Ax_P_Limite := posc.GdX_P_Limite;
Ax_N_Limite := posc.GdX_N_Limite;
Ay_P_Limite := posc.GdY_P_Limite;
Ay_N_Limite := posc.GdY_N_Limite;
Az_P_Limite := posc.GdZ_P_Limite;
Az_N_Limite := posc.GdZ_N_Limite;


DisSensor_SSC1	:= Sensor.sensorD.SSC1_1;
DisSensor_Dis	:= Sensor.sensorD.Distance;

i_Lens_Cap_IsOpen := IO.i515;
i_Lens_Cap_IsClose := IO.i514;


IF (EStop OR SystemError) THEN
	IF bBuzy THEN
		step := step  + 10000;
	END_IF
	IF StepA.bBuzy THEN
		StepA.step := StepA.step  + 10000;
	END_IF
	Hmi_Web.Process_Data_UUID_D_Start := FALSE;
	q_Lens_Blow := FALSE;
END_IF

bBuzy := step > 0 AND step < 10000;
bError := step >= 10000;
IF bBuzy OR bError THEN
	bDone := FALSE;
END_IF

Step_01_DoPayloadList();
Step_02_Do_2nd_in_list();
Step_03_DoLaserAction();



StepA.bBuzy := StepA.step > 0 AND StepA.step < 10000;
StepA.bError := StepA.step >= 10000;
IF StepA.bBuzy OR StepA.bError THEN
	StepA.bDone := FALSE;
END_IF

Step_A_01_MoveToXY();
Step_A_02_FindZ();
Step_A_03_FindY();
Step_A_10_MoveToXY_REF();
Step_A_20_ToStanbyPos();

Timer();

RefPos.X := Ax.Pos - pointRef.X;
RefPos.Y := Ay.Pos - pointRef.Y;
RefPos.Z := Az.Pos - pointRef.Z;

ProjectData.Now_Steel_Payload_D_DataNumberDone := WorkNum;


IF i_Lens_Cap_IsOpen THEN
	q_Lens_Cap_Open := FALSE;
END_IF

IF i_Lens_Cap_IsClose THEN
	q_Lens_Cap_Close := FALSE;
END_IF

io.q309 := q_Lens_Cap_Open;
io.q310 := q_Lens_Cap_Close;

io.q308 := q_Lens_Blow;

_log(name:= 'GroupD', step:= step);
_logA(name:= 'GroupD_Mov', step:= StepA.Step);

METHOD Close_Conver
VAR_INPUT
END_VAR
IF NOT bBuzy THEN
	IF NOT i_Lens_Cap_IsClose THEN
		q_Lens_Cap_Open := FALSE;
		q_Lens_Cap_Close := TRUE;
	ELSE
		q_Lens_Cap_Close := FALSE;
	END_IF
END_IF
END_METHOD

METHOD Do_WorkList : BOOL
VAR_INPUT
END_VAR
bDone := FALSE;

// ============ 紀錄啟動條件 ============
_log.fbJson.StartObject();
_log.fbJson.AddKeyString('MethodName','Do_WorkList');
_log.JsonOutput();
// ======================================



Step := 100;
END_METHOD

METHOD FindZ : BOOL
VAR_INPUT
END_VAR
StepA.bDone := FALSE;

// ============ 紀錄啟動條件 ============
_logA.fbJson.StartObject();
_logA.fbJson.AddKeyString('MethodName','FindZ');
_logA.JsonOutput();
// ======================================





StepA.step := 200;
END_METHOD

METHOD FindZ_Fast : BOOL
VAR_INPUT
END_VAR
StepA.bDone := FALSE;

// ============ 紀錄啟動條件 ============
_logA.fbJson.StartObject();
_logA.fbJson.AddKeyString('MethodName','FindZ_Fast');
_logA.JsonOutput();
// ======================================




StepA.step := 220;
END_METHOD

ACTION Oil:
X_Move := Axis.GdX_total_Move - Axis.GdX_Last_Oil;
Y_Move := Axis.GdY_total_Move - Axis.GdY_Last_Oil;
Z_Move := Axis.GdZ_total_Move - Axis.GdZ_Last_Oil;

IF X_Move > 1000000 OR Y_Move > 1000000 OR Z_Move > 1000000 THEN
	IO.q207 := TRUE;
END_IF
END_ACTION

METHOD Open_Conver
VAR_INPUT
END_VAR
IF NOT bBuzy  THEN
	IF NOT i_Lens_Cap_IsOpen THEN
		q_Lens_Cap_Open := TRUE;
		q_Lens_Cap_Close := FALSE;
	ELSE
		q_Lens_Cap_Open := FALSE;
	END_IF
END_IF
END_METHOD

PROPERTY ReadyToMove : BOOL
GET
ReadyToMove := _ReadyToMove;
END_GET
SET
_ReadyToMove := ReadyToMove;
END_SET
END_PROPERTY

PROPERTY ReadyToPrint : BOOL
GET
ReadyToPrint := _ReadyToPrint;
END_GET
SET
_ReadyToPrint := ReadyToPrint;
END_SET
END_PROPERTY

METHOD Set_X_Ref
VAR_INPUT
	Value : LREAL;
END_VAR
pointRef.X := Value;
END_METHOD

METHOD Set_Y_Ref
VAR_INPUT
	Value : LREAL;
END_VAR
pointRef.Y := Value;
END_METHOD

ACTION Step_01_DoPayloadList:
CASE step OF
(*	===============================================
		開始做 Payload_B_Data_buff 清單內的工作
	===============================================*)
	100: // 以數量判斷是否有工作
		WorkNum := 0;
		IF ProjectData.Now_Steel_Payload_D_DataNumber > 0 THEN
			step := step + 1;
		ELSE
			q_Lens_Cap_Close := TRUE;
			bDone := TRUE;
			Step := 0;
		END_IF
 
			
	101:
		// 初始化工作暫存器
		Hmi_Web.Process_Data_UUID_D_Start := FALSE;
		WorkNum := 0;
		q_Lens_Cap_Open := TRUE;
		step := 110;
		
(*	===============================================
					設定工作中的專案
	===============================================*)
	110:
		ProjectData.Payload_D_Data_Now := ProjectData.Payload_D_Data_buff[WorkNum];
		Hmi_Web.Process_Data_UUID_D := ProjectData.Payload_D_Data_buff[WorkNum].data_uid;
		step := step + 1;
	
	111:
		step := 120;
		
(*	===============================================
					移動到位置
	===============================================*)
	120:
		IF _ReadyToMove THEN
			step := step + 1;
		END_IF
		
	121:
		tmpPos_Y1 := ProjectData.Payload_D_Data_Now.Point_Y;
		
		IF tmpPos_Y1 > 80 AND tmpPos_Y1 < (ProjectData.Now_Steel.Height -80) THEN
			tmpPos_Y1 := tmpPos_Y1 - 2;
		END_IF
		
		XY_Move_Ref(
			ProjectData.Payload_D_Data_Now.Point_X, 
			tmpPos_Y1, 
			SpdC.HighSpeed
		);
		step := step + 1;
		
	122:
		IF stepA.bBuzy OR stepA.bError THEN
			step := step + 1;
		END_IF
		
	123:
		IF stepA.bDone THEN
			step := step + 1;
		ELSIF stepA.bError THEN
			step := step + 10000;
		END_IF
		
	124:
		step := 130;
	

(*	===============================================
				雷射主機 啟動 預覽/雕刻 動作
	===============================================*)	
	130:
		step := 300;
END_CASE
END_ACTION

ACTION Step_02_Do_2nd_in_list:
CASE step OF
	200:
		step := 210;
		
(*	===============================================
					設定工作中的專案
	===============================================*)
	210:
		ProjectData.Payload_D_Data_Now := ProjectData.Payload_D_Data_buff[WorkNum];
		Hmi_Web.Process_Data_UUID_D := ProjectData.Payload_D_Data_buff[WorkNum].data_uid;
		step := step + 1;
	
	211:
		step := 220;
		
(*	===============================================
					移動到位置
	===============================================*)
	220:
		tmpPos_Y1 := ProjectData.Payload_D_Data_Now.Point_Y;
		
		IF tmpPos_Y1 > 80 AND tmpPos_Y1 < (ProjectData.Now_Steel.Height -80) THEN
			tmpPos_Y1 := tmpPos_Y1 - 2;
		END_IF
		
		XY_Move_Ref(
			ProjectData.Payload_D_Data_Now.Point_X, 
			tmpPos_Y1, 
			SpdC.HighSpeed
		);
		step := step + 1;
		
	221:
		IF stepA.bBuzy OR stepA.bError THEN
			step := step + 1;
		END_IF
		
	222:
		IF stepA.bDone THEN
			step := step + 1;
		ELSIF stepA.bError THEN
			step := step + 10000;
		END_IF
		
	223:
		step := 230;

(*	===============================================
				雷射主機 啟動 預覽/雕刻 動作
	===============================================*)	
	230:
		step := 300;
		
END_CASE
END_ACTION

ACTION Step_03_DoLaserAction:
CASE step OF
	300:
		IF ReadyToPrint THEN
			step := step + 1;
		END_IF
		
	301:
		sql_hand := ReadSQLData.Set_Payload_Start(ProjectData.Payload_D_Data_Now.data_uid);
		IF sql_hand <> 0 THEN
			step := step + 1;
		END_IF
		
	302:
		step := 310;

(*	===============================================
				雷射主機 啟動 預覽/雕刻 動作
	===============================================*)	
	310:
		q_Lens_Blow := TRUE;
		q_Lens_Cap_Open := TRUE;
		IF LEN(Hmi_Web.Process_Data_UUID_D) = 0 THEN
			Hmi_Web.Process_Data_UUID_D := ProjectData.Payload_D_Data_buff[WorkNum].data_uid;
		ELSE
			step := step + 1;
		END_IF
		
	311: // 確認鏡頭蓋已開
		IF i_Lens_Cap_IsOpen THEN
			step := step + 1;
		END_IF
		
	312:
		Hmi_Web.Process_Data_UUID_D_Start := TRUE;
		// ============ 紀錄啟動條件 ============
		_log.fbJson.StartObject();
		_log.fbJson.AddKeyString('StepName','Laser_D_Start');
		_log.fbJson.AddKeyBool('Process_Data_UUID_D_Start', Hmi_Web.Process_Data_UUID_A_Start);
		_log.fbJson.AddKeyString('Payload_D_Data_Now', ProjectData.Payload_D_Data_Now.data_uid);
		_log.JsonOutput();
		// ======================================
		step := step + 1;
		
	313:	
		tmr01.PT := T#500MS;
		tmr01.IN := TRUE;
		IF tmr01.Q THEN
			tmr01.IN := FALSE;
			tmr02.IN := FALSE;
			step := step + 1;
		END_IF
		
	314:
		tmr01.PT := TO_TIME(MaCfg.LaserPrinter_Timeout);
		tmr01.IN := TRUE;
		tmr02.PT := T#250MS;
		tmr02.IN := NOT Hmi_Web.Process_Data_UUID_D_Start;
		
		IF tmr02.q THEN // 程式通知打標完成
			Hmi_Web.Process_Data_UUID_D :='';
			tmr01.IN := FALSE;
			tmr02.IN := FALSE;
			// ============ 紀錄啟動條件 ============
			_log.fbJson.StartObject();
			_log.fbJson.AddKeyString('StepName','Laser_D_Done');
			_log.JsonOutput();
			// ======================================
			step := step + 1;
		ELSIF tmr01.Q THEN // 打標超時
			tmr01.IN := FALSE;
			tmr02.IN := FALSE;
			pMsg.Push_Error("GroupD:雷射動作超時");
			step := step + 10000;
		END_IF

	
	315:
		q_Lens_Blow := FALSE;
		WorkNum := WorkNum + 1;
		step := 320;
		
(*	================================================
				開始下個循環或此區域結束
	================================================*)	
	320:
		sql_hand := ReadSQLData.Set_Payload_Finish(ProjectData.Payload_D_Data_Now.data_uid);
		IF sql_hand <> 0 THEN
			step := step + 1;
		END_IF
		
	321:
		IF WorkNum < ProjectData.Now_Steel_Payload_D_DataNumber THEN
		// 這個區域還有工作
			step := step + 1;
		ELSE
		// 這個區域工作結束
			step := 390;
		END_IF
		
	322:
		// 設定工作中的專案
		step := 200;
		
(*	========================================
				這個區域工作結束
	========================================*)		
	390:
		 // 關 鏡頭蓋
		q_Lens_Cap_Close := TRUE;
		
		bDone := TRUE;
		step := 0;
END_CASE
END_ACTION

ACTION Step_A_01_MoveToXY:
CASE StepA.step OF
	100:
		IF moveCmd_X < Ax_P_Limite AND moveCmd_X > Ax_N_Limite THEN
			StepA.step := StepA.step + 1;
		ELSIF moveCmd_X >= Ax_P_Limite THEN
			StepA.step := StepA.step + 10000;
			pMsg.Push_Alarm("GroupA MoveXY:命令位置超出X軸+極限");
		ELSE
			StepA.step := StepA.step + 10000;
			pMsg.Push_Alarm("GroupA MoveXY:命令位置超出X軸-極限");
		END_IF
 
			
	101:
		IF moveCmd_Y < Ay_P_Limite AND moveCmd_Y > Ay_N_Limite THEN
			StepA.step := StepA.step + 1;
		ELSIF moveCmd_Y >= Ay_P_Limite THEN
			StepA.step := StepA.step + 10000;
			pMsg.Push_Alarm("GroupA MoveXY:命令位置超出Y軸+極限");
		ELSE
			StepA.step := StepA.step + 10000;
			pMsg.Push_Alarm("GroupA MoveXY:命令位置超出Y軸-極限");
		END_IF
		
	102:
		StepA.step := 110;
		
	110:
		Ax.AbsMove(moveCmd_X, moveCmd_Spd);
		Ay.AbsMove(moveCmd_Y, moveCmd_Spd);
		StepA.step := StepA.step + 1;
		
	111:
		IF (Axs.bBuzy OR Axs.bError) AND (Ays.bBuzy OR Ays.bError) THEN
			StepA.step := StepA.step + 1;
		END_IF
		
	112:
		IF Axs.bDone AND Ays.bDone THEN
			StepA.step := StepA.step + 1;
		ELSIF Axs.bError OR Ays.bError THEN
			StepA.step := StepA.step + 10000;
		END_IF
		
	113:
		StepA.bDone := TRUE;
		StepA.step := 0;
		
END_CASE
END_ACTION

ACTION Step_A_02_FindZ:
CASE StepA.step OF
	200: // 判斷當距離再200~400間
		IF DisSensor_Dis < 200 OR DisSensor_Dis > 400 THEN
			StepA.step := StepA.step + 1;
		ELSE
			StepA.step := 220;
		END_IF
		
	201:
		StepA.step := 210;
		
	210: 
		q_Lens_Cap_Open := TRUE;
		StepA.step := StepA.step + 1;
		
	211:
		StepA.step := 220;
		
	220:
		tmpPos_X := 0;
		
		IF ProjectData.Now_Steel.Width < 200 THEN
			tmpPos_Y := MaCfg.laserD_Y_ReferencePos + (ProjectData.Now_Steel.Height / 2);
		ELSE
			tmpPos_Y := MaCfg.laserD_Y_ReferencePos + 75;
		END_IF
			
		tmpPos_Z := MaCfg.laserD_Dis - (ProjectData.Now_Steel.Width / 2);
		IF tmpPos_Z < 20 THEN
			pMsg.Push_Error(WStrConcat(
				"GroupD_Find_Z:Z軸計算位置錯誤 pos:",
				TO_WSTRING(tmpPos_Z)
			));
		END_IF
		StepA.step := StepA.step + 1;
		
	221: 
		Ax.AbsMove(tmpPos_X, SpdC.HighSpeed);
		Ay.AbsMove(tmpPos_Y, SpdC.HighSpeed);
		Az.AbsMove(tmpPos_Z , SpdC.HighSpeed);
		StepA.step := StepA.step + 1;
		
	222:
		IF (Axs.bBuzy OR Axs.bError) AND (Ays.bBuzy OR Ays.bError) AND (Azs.bBuzy OR Azs.bError) THEN
			StepA.step := StepA.step + 1;
		END_IF
		
	223:
		IF Axs.bDone AND Ays.bDone AND Azs.bDone THEN
			StepA.step := StepA.step + 1;
		ELSIF Axs.bError OR Ays.bError THEN
			StepA.step := StepA.step + 10000;
		END_IF
		
	224:
		q_Lens_Cap_Open := TRUE;
		StepA.step := 230;
		
		
	230:
		IF DisSensor_Dis > 1 THEN
			moveZdis := DisSensor_Dis - Macfg.laserD_Dis;
			StepA.step := StepA.step + 1;
		ELSE
			tmpPos_X := tmpPos_X + 15;
			StepA.step := 221;
		END_IF
		
	231:
		Az.RelMove(moveZdis * -1, SpdC.HighSpeed);
		StepA.step := StepA.step + 1;
		
	232:
		IF GdZ.bBuzy OR GdZ.bError THEN
			StepA.step := StepA.step + 1;
		END_IF
		
	233:
		IF GdZ.bDone THEN
			StepA.step := StepA.step + 1;
		ELSIF GdZ.bError THEN
			StepA.step := StepA.step + 10000;
		END_IF
		
	234:
		tmr01A.IN := TRUE;
		tmr01A.PT := T#2S;
		IF tmr01A.Q THEN
			tmr01A.IN := FALSE;
			StepA.step := StepA.step + 1;
		END_IF
		
	235:
		StepA.step := 240;
		
		
	240:
		moveZdis := DisSensor_Dis - Macfg.laserD_Dis;
		StepA.step := StepA.step + 1;
		
	241:
		Az.RelMove(moveZdis * -1, SpdC.LowSpeed);
		StepA.step := StepA.step + 1;
		
	242:
		IF GdZ.bBuzy OR GdZ.bError THEN
			StepA.step := StepA.step + 1;
		END_IF
		
	243:
		IF GdZ.bDone THEN
			StepA.step := StepA.step + 1;
		ELSIF GdZ.bError THEN
			StepA.step := StepA.step + 10000;
		END_IF
		
	244:
		StepA.step := 250;
		
	250:
		q_Lens_Cap_Open := FALSE;
		z_PosMeasure := Az.Pos;
		StepA.bDone := TRUE;
		StepA.step	:= 0;
		
END_CASE
END_ACTION

ACTION Step_A_03_FindY:
CASE StepA.step OF
	300: // 判斷當距離再200~400間，才做偵測
		IF DisSensor_Dis > 200 OR DisSensor_Dis < 400 THEN
			StepA.step := StepA.step + 1;
		ELSE
			pmsg.Push_Alarm_NoPause("GroupD:Z軸距離感應器不再感應範圍內，取消Y軸原點偵測，使用預設值");
			StepA.step	:= 380;
		END_IF
		
	301:
		StepA.step := 310;
		
	310: 
		Ay.AbsMove(100, 50);
		StepA.step := StepA.step + 1;
		
	311:
		IF Ays.bBuzy OR Ays.bError THEN
			StepA.step := StepA.step + 1;
		END_IF
		
	312:
		IF NOT DisSensor_SSC1 THEN
			Ay.Stop();
			StepA.step := StepA.step + 1;
		ELSIF Ays.bDone THEN
			pmsg.Push_Alarm_NoPause("GroupD:Z軸距離感應器訊號錯誤");
			StepA.step := 380;
		ELSIF Ays.bError THEN
			StepA.step := StepA.step + 10000;
		END_IF
		
	313:
		tmr01A.IN := TRUE;
		tmr01A.PT := T#500MS;
		IF tmr01A.Q THEN
			tmr01A.IN := FALSE;
			StepA.step := StepA.step + 1;
		END_IF
		
	314:
		StepA.step := 320;
		
	320:
		Ay.AbsMove(Ay_P_Limite - 5, 5);
		StepA.step := StepA.step + 1;
		
	321:
		IF (Ays.bBuzy OR Ays.bError) THEN
			StepA.step := StepA.step + 1;
		END_IF
		
	322:
		IF DisSensor_SSC1 THEN
			Ay.Stop();
			StepA.step := StepA.step + 1;
		ELSIF Ays.bDone THEN
			pmsg.Push_Alarm_NoPause("GroupD:Z軸距離感應器訊號錯誤");
			StepA.step := 380;
		ELSIF Ays.bError THEN
			StepA.step := StepA.step + 10000;
		END_IF
		
	323:
		tmr01A.IN := TRUE;
		tmr01A.PT := T#500MS;
		IF tmr01A.Q THEN
			tmr01A.IN := FALSE;
			StepA.step := StepA.step + 1;
		END_IF
		
	324:
		StepA.step := 330;
		
		
	330:
		Ay.AbsMove(100, 0.5);
		StepA.step := StepA.step + 1;
		
	331:
		IF Ays.bBuzy OR Ays.bError THEN
			StepA.step := StepA.step + 1;
		END_IF
		
	332:
		IF NOT DisSensor_SSC1 THEN
			Ay.Stop();
			StepA.step := StepA.step + 1;
		ELSIF Ays.bDone THEN
			pmsg.Push_Alarm_NoPause("GroupD:Z軸距離感應器訊號錯誤");
			StepA.step := 380;
		ELSIF Ays.bError THEN
			StepA.step := StepA.step + 10000;
		END_IF
		
	333:
		tmr01A.IN := TRUE;
		tmr01A.PT := T#500MS;
		IF tmr01A.Q THEN
			tmr01A.IN := FALSE;
			StepA.step := StepA.step + 1;
		END_IF
		
	334:
		StepA.step := 340;
		
		
	340:
		Set_Y_Ref(Ay.Pos);
		StepA.step := StepA.step + 1;
		
	341:
		StepA.step := 390;
		
	
	380:
		IF projectData.Now_Steel.Height > 0 THEN
			Set_Y_Ref(Ay_P_Limite + 56 - projectData.Now_Steel.Height);
		ELSE
			Set_Y_Ref(Ay_P_Limite + 56 - 500);
		END_IF
		StepA.step := StepA.step + 1;
		
	381:
		StepA.step	:= 390;
	
	390:
		z_PosMeasure := GaZ.Pos;
		StepA.bDone := TRUE;
		StepA.step	:= 0;
		
END_CASE
END_ACTION

ACTION Step_A_10_MoveToXY_REF:
CASE StepA.step OF
	1000:// 計算相對距離
		tmpPos_X := moveCmd_X - pointRef.X;
		tmpPos_Y := moveCmd_Y + pointRef.Y;
		Dxf_Y_Move := 0;
		StepA.step := StepA.step + 1;
		
	1001:
		IF tmpPos_X < Ax_P_Limite AND tmpPos_X > Ax_N_Limite THEN
			StepA.step := StepA.step + 1;
		ELSIF tmpPos_X >= Ax_P_Limite THEN
			StepA.step := StepA.step + 10000;
			pMsg.Push_Alarm("GroupD MoveXY:命令位置超出X軸+極限");
		ELSE
			StepA.step := StepA.step + 10000;
			pMsg.Push_Alarm("GroupD MoveXY:命令位置超出X軸-極限");
		END_IF
 
			
	1002:
		IF tmpPos_Y < Ay_P_Limite AND tmpPos_Y > Ay_N_Limite THEN
			StepA.step := StepA.step + 1;
		ELSIF tmpPos_Y >= Ay_P_Limite THEN
			StepA.step := StepA.step + 10000;
			pMsg.Push_Alarm("GroupD MoveXY_Ref:命令位置超出Y軸+極限");
		ELSE
			StepA.step := StepA.step + 10000;
			pMsg.Push_Alarm("GroupD MoveXY_Ref:命令位置超出Y軸-極限");
		END_IF
		
	1003:
		StepA.step := 1010;
		
	1010:
		Ax.AbsMove(tmpPos_X, moveCmd_Spd);
		Ay.AbsMove(tmpPos_Y, moveCmd_Spd);
		StepA.step := StepA.step + 1;
		
	1011:
		IF (Axs.bBuzy OR Axs.bError) AND (Ays.bBuzy OR Ays.bError) THEN
			StepA.step := StepA.step + 1;
		END_IF
		
	1012:
		IF Axs.bDone AND Ays.bDone THEN
			StepA.step := StepA.step + 1;
		ELSIF Axs.bError OR Ays.bError THEN
			StepA.step := StepA.step + 10000;
		END_IF
		
	1013:
		tmr01A.IN := TRUE;
		tmr01A.PT := T#1S;
		IF tmr01A.Q THEN
			tmr01A.IN := FALSE;
			StepA.step := StepA.step + 1;
		END_IF
		
	1014:
		StepA.step := 1020;
		
	1020:
		StepA.bDone := TRUE;
		StepA.step := 0;
		
END_CASE
END_ACTION

ACTION Step_A_20_ToStanbyPos:
CASE StepA.step OF
	2000:
		q_Lens_Cap_Close := TRUE;
		StepA.step := 2010;
		
	2010:
		IF Az.Pos > posc.pos_GdZ_stanby - 20 THEN
			StepA.step := 2020;
		ELSE
			StepA.step := StepA.step + 1;
		END_IF
		
	2011:
		Az.RelMove(20, SpdC.HomeSpeed);
		StepA.step := StepA.step + 1;
		
	2012:
		IF Azs.bDone OR Azs.bError OR NOT GdZ.outLimiter THEN
			StepA.step := StepA.step + 1;
		END_IF
		
	2013:
		IF Azs.bDone THEN
			StepA.step := StepA.step + 1;
		ELSIF Azs.bError THEN
			StepA.step := StepA.step + 10000;
		END_IF
		
	2014:
		StepA.step := 2020;
		
	2020:
		Ax.AbsMove(posc.pos_GdX_stanby, moveCmd_Spd);
		StepA.step := StepA.step + 1;
		
	2021:
		IF (Axs.bBuzy OR Axs.bError) THEN
			StepA.step := StepA.step + 1;
		END_IF
		
	2022:
		IF Axs.bDone THEN
			StepA.step := StepA.step + 1;
		ELSIF Axs.bError THEN
			StepA.step := StepA.step + 10000;
		END_IF
	
	2023:
		StepA.step := 2030;
	
	2030:
		Ay.AbsMove(posc.pos_GdY_stanby, moveCmd_Spd);
		Az.AbsMove(posc.pos_GdZ_stanby, moveCmd_Spd);
		StepA.step := StepA.step + 1;
		
	2031:
		IF (Azs.bBuzy OR Azs.bError) AND (Ays.bBuzy OR Ays.bError)  THEN
			StepA.step := StepA.step + 1;
		END_IF
		
	2032:
		IF Azs.bDone AND Ays.bDone THEN
			StepA.step := StepA.step + 1;
		ELSIF Azs.bError OR Ays.bError THEN
			StepA.step := StepA.step + 10000;
		END_IF
		
	2033:
		StepA.step := 2040;
		
		
	2040:
		StepA.bDone := TRUE;
		StepA.step := 0;
		
END_CASE
END_ACTION

ACTION Timer:
tmr01A();
tmr01();
tmr02();

// tmr_oil(in := IO.q207 AND IO.i310, PT:=T#2S);
tmr_oil(in := IO.q207, PT:=T#2S);

IF tmr_oil.Q THEN
	IO.q207 := FALSE;
	
	Axis.GdX_Last_Oil := Axis.GdX_total_Move;
	
	Axis.GdY_Last_Oil := Axis.GdY_total_Move;
	
	Axis.GdZ_Last_Oil := Axis.GdZ_total_Move;
END_IF
END_ACTION

METHOD ToStanby : BOOL
VAR_INPUT
	Speed : LREAL := 0;
END_VAR
StepA.bDone := FALSE;
IF Speed > 0 THEN
	moveCmd_Spd := Speed;
ELSE
	moveCmd_Spd := SpdC.HomeSpeed;
END_IF

// ============ 紀錄啟動條件 ============
_logA.fbJson.StartObject();
_logA.fbJson.AddKeyString('MethodName','ToStanby');
_logA.fbJson.AddKeyLreal('Velocity', Speed);
_logA.JsonOutput();
// ======================================




StepA.step := 2000;
END_METHOD

METHOD XY_Move : BOOL
VAR_INPUT
	X_Point : LREAL;
	Y_Point	: LREAL;
	Speed : LREAL;
END_VAR
moveCmd_X := X_Point;
moveCmd_Y := Y_Point;
moveCmd_Spd := Speed;

StepA.bDone := FALSE;

// ============ 紀錄啟動條件 ============
_logA.fbJson.StartObject();
_logA.fbJson.AddKeyString('MethodName','XY_Move');
_logA.fbJson.AddKeyLreal('X_Point', X_Point);
_logA.fbJson.AddKeyLreal('Y_Point', Y_Point);
_logA.fbJson.AddKeyLreal('Velocity', Speed);
_logA.JsonOutput();
// ======================================


StepA.step := 100;
END_METHOD

METHOD XY_Move_Ref : BOOL
VAR_INPUT
	X_Point : LREAL;
	Y_Point	: LREAL;
	Speed : LREAL;
END_VAR
moveCmd_X := X_Point;
moveCmd_Y := Y_Point;
moveCmd_Spd := Speed;

StepA.bDone := FALSE;

// ============ 紀錄啟動條件 ============
_logA.fbJson.StartObject();
_logA.fbJson.AddKeyString('MethodName','XY_Move_Ref');
_logA.fbJson.AddKeyLreal('X_Point', X_Point);
_logA.fbJson.AddKeyLreal('Y_Point', Y_Point);
_logA.fbJson.AddKeyLreal('Velocity', Speed);
_logA.JsonOutput();
// ======================================


StepA.step := 1000;
END_METHOD

END_PROGRAM

// ---- POUs/動作流程控制/測試功能/TestActionPou.TcPOU
PROGRAM TestActionPou
VAR
	// 步驟
	Step: INT;
	// 已執行的清單
	ActionStep: UINT;
	
	
	
	
	
	// 選擇的軸
	AxisSelect: INT;
	// 移動的位置
	MovePos: REAL;
	// 移動的速度
	MoveSpeed: REAL;
	
	// 清單重置用
	i: INT;
	tmr1: TON;
END_VAR

IF (EStop OR SystemError) THEN
	Step := 0;
END_IF

Step00_ActionSelect();

Step01_Move();

ACTION Step00_ActionSelect:
CASE Step OF
	1:
		ActionStep := 0;
		FOR i := 0 TO 10 DO
			AxisTest.test_Action_List[i].Cycles_Done := 0;
		END_FOR
		Step := Step + 1;
		
	2:
		Step := 10;
	
	10:
		CASE AxisTest.test_Action_List[ActionStep].ActionSelect OF
			1: // 軸移動
				Step := 100;
				
			2: // 等待移動完成
				Step := 200;
				
			3:// 等待時間
				tmr1.PT := REAL_TO_TIME(AxisTest.test_Action_List[ActionStep].WaitTime*1000);
				Step := 300;
				
			4:// 重複
				Step := 400;
				
			ELSE
				Step := 0;
		END_CASE
		
		
	200:
		IF NOT GaX.bBuzy AND NOT GaY.bBuzy AND NOT GaZ.bBuzy AND 
			NOT GbX.bBuzy AND NOT GbY.bBuzy AND NOT GbZ.bBuzy AND 
			NOT GcX.bBuzy AND NOT GcY.bBuzy AND NOT GcZ.bBuzy AND 
			NOT GdX.bBuzy AND NOT GdY.bBuzy AND NOT GdZ.bBuzy AND 
			NOT Fx.bBuzy  
		THEN
			Step := 900;
		END_IF
		
	300:
		tmr1.IN :=TRUE;
		IF tmr1.Q THEN
			tmr1.IN := FALSE;
			Step := Step + 1;
		END_IF
		
	301:
		Step := 900;
		
	400:
		IF AxisTest.test_Action_List[ActionStep].Cycles_Done >= AxisTest.test_Action_List[ActionStep].Cycles THEN
			Step := Step + 1;
		ELSE
			AxisTest.test_Action_List[ActionStep].Cycles_Done := AxisTest.test_Action_List[ActionStep].Cycles_Done + 1;
			ActionStep := AxisTest.test_Action_List[ActionStep].Cycles_StartStep;
			Step := 10;
		END_IF 
		
	401:
		Step := 900;
		
	900:
		IF ActionStep <= 10 THEN
			ActionStep := ActionStep + 1;
			Step := 10;
		ELSE
			Step := 0;
		END_IF
END_CASE

tmr1();
END_ACTION

ACTION Step01_Move:
CASE Step OF
	100:
		AxisSelect := AxisTest.test_Action_List[ActionStep].AxisSelect;
		MovePos := AxisTest.test_Action_List[ActionStep].Pos;
		MoveSpeed := AxisTest.test_Action_List[ActionStep].Speed;
		
		Step := Step + 1;
	
	101:
		CASE AxisSelect OF
			1:
				IF NOT GaX.bBuzy THEN
					Step := Step + 1;
				END_IF
				
			2:
				IF NOT GaY.bBuzy THEN
					Step := Step + 1;
				END_IF
				
			3:
				IF NOT GaZ.bBuzy THEN
					Step := Step + 1;
				END_IF
				
			11:
				IF NOT GbX.bBuzy THEN
					Step := Step + 1;
				END_IF
				
			12:
				IF NOT GbY.bBuzy THEN
					Step := Step + 1;
				END_IF
				
			13:
				IF NOT GbZ.bBuzy THEN
					Step := Step + 1;
				END_IF
				
			21:
				IF NOT GcX.bBuzy THEN
					Step := Step + 1;
				END_IF
				
			22:
				IF NOT GcY.bBuzy THEN
					Step := Step + 1;
				END_IF
				
			23:
				IF NOT GcZ.bBuzy THEN
					Step := Step + 1;
				END_IF
				
			31:
				IF NOT GdX.bBuzy THEN
					Step := Step + 1;
				END_IF
				
			32:
				IF NOT GdY.bBuzy THEN
					Step := Step + 1;
				END_IF
				
			33:
				IF NOT GdZ.bBuzy THEN
					Step := Step + 1;
				END_IF
				
			41:
				IF NOT Fx.bBuzy THEN
					Step := Step + 1;
				END_IF
		END_CASE
		
		
	102:
		CASE AxisSelect OF
			1:
				GaX.AbsMove(MovePos, MoveSpeed);
				IF GaX.bBuzy THEN
					Step := Step + 1;
				END_IF
				
			2:
				GaY.AbsMove(MovePos, MoveSpeed);
				IF GaY.bBuzy THEN
					Step := Step + 1;
				END_IF
				
			3:
				GaZ.AbsMove(MovePos, MoveSpeed);
				IF GaZ.bBuzy THEN
					Step := Step + 1;
				END_IF
				
			11:
				GbX.AbsMove(MovePos, MoveSpeed);
				IF GbX.bBuzy THEN
					Step := Step + 1;
				END_IF
				
			12:
				GbY.AbsMove(MovePos, MoveSpeed);
				IF GbY.bBuzy THEN
					Step := Step + 1;
				END_IF
				
			13:
				GbZ.AbsMove(MovePos, MoveSpeed);
				IF GbZ.bBuzy THEN
					Step := Step + 1;
				END_IF
				
			21:
				GcX.AbsMove(MovePos, MoveSpeed);
				IF GcX.bBuzy THEN
					Step := Step + 1;
				END_IF
				
			22:
				GcY.AbsMove(MovePos, MoveSpeed);
				IF GcY.bBuzy THEN
					Step := Step + 1;
				END_IF
				
			23:
				GcZ.AbsMove(MovePos, MoveSpeed);
				IF GcZ.bBuzy THEN
					Step := Step + 1;
				END_IF
				
			31:
				GdX.AbsMove(MovePos, MoveSpeed);
				IF GdX.bBuzy THEN
					Step := Step + 1;
				END_IF
				
			32:
				GdY.AbsMove(MovePos, MoveSpeed);
				IF GdY.bBuzy THEN
					Step := Step + 1;
				END_IF
				
			33:
				GdZ.AbsMove(MovePos, MoveSpeed);
				IF GdZ.bBuzy THEN
					Step := Step + 1;
				END_IF
				
			41:
				Fx.AbsMove(MovePos, MoveSpeed);
				IF Fx.bBuzy THEN
					Step := Step + 1;
				END_IF
		END_CASE
		
	103:
		
		Step := 900;
END_CASE
END_ACTION

END_PROGRAM

// ---- POUs/動作流程控制/外部輸送滾輪/ExpConver.TcPOU
{attribute 'TcContextName':='PlcTask'}
PROGRAM ExpConver
VAR
(*	======================================================
					外部輸送機 訊號輸出
	======================================================*)
	// 進料機 動作中
	Feed_bBuzy						AT %I*	: BOOL;
	// 進料機 動作完成
	Feed_bDone 						AT %I*	: BOOL;
	// 進料機 發生錯誤
	Feed_bError 					AT %I*	: BOOL;
	
	// 進料材料寬度
	Feed_Workpiace_W 				AT %I*	: LREAL;
	
	// 進料材料高度
	Feed_Workpiace_H 				AT %I*	: LREAL;
	
	// 執行中的動作
	ActionMode_Now 					AT %I*	: UINT;
	
	
	
	// 靠邊 動作中
	PullOver_bBuzy					AT %I*	: BOOL;
	// 靠邊  動作完成
	PullOver_bDone 					AT %I*	: BOOL;
	// 靠邊  發生錯誤
	PullOver_bError 				AT %I*	: BOOL;
	
	
	// 入料測感應器
	In_sensor 						AT %I*	: WORD;
	
	// 出料測感應器
	Out_sensor 						AT %I*	: WORD;
	
	// 進料滾輪啟動
	In_Moter_Running 				AT %I*	: BOOL;
	// 進料滾輪錯誤
	In_Moter_Error 					AT %I*	: BOOL;
	
	// 出料滾輪啟動
	Out_Moter_Running 				AT %I*	: BOOL;
	// 出料滾輪錯誤
	Out_Moter_Error 				AT %I*	: BOOL;
	
	
(*	======================================================
					外部輸送機 訊號輸入
	======================================================*)
	// 進料機 執行
	ExpConver_Start					AT %Q*	: BOOL;
	
	// 進料機 模式
	ExpConver_Enable				AT %Q*	: BOOL;
	
	// 進料機 模式
	ExpConver_Mode					AT %Q*	: INT;
	
	// 進料機 進料的專案UUID
	ExpConver_WorkOrder_UUID		AT %Q*	: STRING(36);
	
	// 進料機 錯誤重置
	ExpConver_Reset					AT %Q*	: BOOL;
	
	// 靠邊 模式執行
	PullOver_Start					AT %Q*	: BOOL;
	
	// 進料滾輪啟動
	In_Moter_Start 					AT %Q*	: BOOL;
	
	// 出料滾輪啟動
	Out_Moter_Start 				AT %Q*	: BOOL;
	
	trig1: R_TRIG;
	trig2: R_TRIG;
END_VAR

IF (EStop OR SystemError) THEN
	In_Moter_Start := FALSE;
	Out_Moter_Start := FALSE;
	ExpConver_Reset := TRUE;
	ExpConver_Mode := 0;
END_IF

trig2(CLK := Feed_bBuzy );

IF trig2.q THEN
	ExpConver_Start := FALSE;
END_IF

ExpConver_WorkOrder_UUID := Hmi_Web.Auto_ProjectWorkOrder_uuid; 

trig1(CLK := Feed_bError OR Feed_bDone);
IF trig1.Q THEN
	ExpConver_Mode := 0;
END_IF

IF ExpConver_Reset AND ActionMode_Now = 0 AND 
		NOT (EStop OR SystemError) THEN
	ExpConver_Reset := FALSE;
END_IF

IF PullOver_bBuzy THEN
	PullOver_Start := FALSE;
END_IF

ExpConver_Enable := NOT IO.i711 AND NOT( AutoMain.step > 600 AND AutoMain.step < 800 );

METHOD Feed_holding_2_waitLoading
VAR_INPUT
END_VAR
ExpConver_Mode := 0;

ExpConver_Start := TRUE;
END_METHOD

METHOD Feed_PullOver
VAR_INPUT
END_VAR
ExpConver_Mode := 2000;

ExpConver_Start := TRUE;
END_METHOD

METHOD Feed_Reset
VAR_INPUT
END_VAR
ExpConver_Reset := true;
END_METHOD

METHOD FeedAutoStart
VAR_INPUT
END_VAR
ExpConver_Mode := 0;


ExpConver_Start := TRUE;
END_METHOD

METHOD FeedHomeStart
VAR_INPUT
END_VAR
ExpConver_Mode := 100;

ExpConver_Start := TRUE;
END_METHOD

METHOD FeedJogExit
VAR_INPUT
END_VAR
ExpConver_Mode := 8001;

ExpConver_Start := TRUE;
END_METHOD

METHOD FeedJogStart
VAR_INPUT
END_VAR
ExpConver_Mode := 8000;

ExpConver_Start := TRUE;
END_METHOD

METHOD InRollerStart
VAR_INPUT
END_VAR
In_Moter_Start := TRUE;
END_METHOD

METHOD InRollerStop
VAR_INPUT
END_VAR
In_Moter_Start := false;
END_METHOD

METHOD OutRollerStart
VAR_INPUT
END_VAR
Out_Moter_Start := TRUE;
END_METHOD

METHOD OutRollerStop
VAR_INPUT
END_VAR
Out_Moter_Start := false;
END_METHOD

END_PROGRAM

// ---- POUs/硬體控制/其他控制/按鈕燈/Button.TcPOU
PROGRAM Button
VAR
	// 系統開機指示燈
	_SystemPowerButton_Light : USINT := 1;
	// 程式開始指示燈
	_StartButton_Light : USINT;
	// 程式暫停指示燈
	_StopButton_Light : USINT;
	// 程式暫停指示燈
	_ResetButton_Light : USINT;
	// 原點指示燈
	_HomeButton_Light : USINT;
	// 手動模式指示燈
	_JogButtonLight : USINT; 
	// 單節模式指示燈
	_StepModeButtonLight : USINT; 
	// 自動模式指示燈
	_AutoModeButtonLight : USINT; 
	
	pc_Shutdown: NT_Shutdown;
	pc_AbortShutdown: NT_AbortShutdown;
	pc_Shutdown2: NT_Shutdown;
	pc_AbortShutdown2: NT_AbortShutdown;
	flash_clk: BOOL;
	jogbtn_trig: R_TRIG;
	StepButton: R_TRIG;
	StartButton_LDP: F_TRIG;
	SystemPowerButton_Ldp: R_TRIG;
END_VAR

VAR_OUTPUT
	// 系統電源
	SystemPowerButton : BOOL;
	// 程式開始
	StartButton : BOOL;
	// 程式暫停
	StopButton : BOOL;
	// 重置
	ResetButton : BOOL;
	// 原點
	HomeButton : BOOL;
	// 手動模式
	JogButton : BOOL; 
	// 單節模式
	StepModeButton : BOOL; 
	// 自動模式
	AutoModeButton : BOOL; 
END_VAR

SystemPowerButton	:= IO.i102;
StartButton			:= IO.i104;
StopButton			:= IO.i103;
ResetButton			:= IO.i105;
HomeButton			:= IO.i106;
JogButton			:= IO.i108;
StepModeButton		:= IO.i109;
AutoModeButton		:= IO.i110;

flash_clk := LightTower.clk;


CASE _SystemPowerButton_Light OF
	0:
		io.q101 := FALSE;
	
	1:
		io.q101 := TRUE;
		
	2:
		io.q101 := flash_clk;
END_CASE

CASE _StopButton_Light OF
	0:
		io.q102 := FALSE;
	
	1:
		io.q102 := TRUE;
		
	2:
		io.q102 := flash_clk;
END_CASE

CASE _StartButton_Light OF
	0:
		io.q103 := FALSE;
	
	1:
		io.q103 := _StopButton_Light = 0;
		
	2:
		io.q103 := _StopButton_Light = 0 and flash_clk;
END_CASE


CASE _ResetButton_Light OF
	0:
		io.q104 := FALSE;
	
	1:
		io.q104 := TRUE;
		
	2:
		io.q104 := flash_clk;
END_CASE


CASE _HomeButton_Light OF
	0:
		io.q105 := FALSE;
	
	1:
		io.q105 := TRUE;
		
	2:
		io.q105 := flash_clk;
END_CASE


CASE _JogButtonLight OF
	0:
		io.q107 := FALSE;
	
	1:
		io.q107 := TRUE;
		
	2:
		io.q107 := flash_clk;
END_CASE


CASE _StepModeButtonLight OF
	0:
		io.q108 := FALSE;
	
	1:
		io.q108 := TRUE;
		
	2:
		io.q108 := flash_clk;
END_CASE

CASE _AutoModeButtonLight OF
	0:
		io.q109 := FALSE;
	
	1:
		io.q109 := TRUE;
		
	2:
		io.q109 := flash_clk;
END_CASE

PowerButtonAction();
StartButtonAction();
ResetButtonAction();


HomeButtonAction();
JogButtonAction();

ACTION AutoModeButtonAction:
IF AutoMain.step = 0 OR AutoMain.step > 2000 THEN
	Button.AutoModeButtonLight := 0;
END_IF
END_ACTION

PROPERTY AutoModeButtonLight : USINT
GET
AutoModeButtonLight := _AutoModeButtonLight;
END_GET
SET
_AutoModeButtonLight := AutoModeButtonLight;
END_SET
END_PROPERTY

PROPERTY HomeButton_Light : USINT
GET
HomeButton_Light := _HomeButton_Light;
END_GET
SET
_HomeButton_Light := HomeButton_Light;
END_SET
END_PROPERTY

ACTION HomeButtonAction:
IF HomeButton THEN
	IF NOT AutoMain.bBuzy THEN
		AutoMain.Homming();
	END_IF
END_IF
END_ACTION

ACTION JogButtonAction:
IF AutoMain.step >= 8000 AND AutoMain.step < 8100 THEN
	Button.JogButtonLight := 1;
ELSIF AutoMain.step >= 8100 AND AutoMain.step < 9800 THEN
	Button.JogButtonLight := 2;
ELSE
	Button.JogButtonLight := 0;
END_IF


jogbtn_trig(CLK := JogButton);
IF jogbtn_trig.Q THEN
	IF AutoMain.step = 0 THEN
		AutoMain.JogMode();
	ELSIF AutoMain.step = 8001 THEN
		AutoMain.JogMode_Exit();
	END_IF
END_IF
END_ACTION

PROPERTY JogButtonLight : USINT
GET
JogButtonLight := _JogButtonLight;
END_GET
SET
_JogButtonLight := JogButtonLight;
END_SET
END_PROPERTY

ACTION PowerButtonAction:
SystemPowerButton_Ldp(CLK:=SystemPowerButton);


IF SystemPowerButton_Ldp.Q THEN
	IF SystemPowerButton_Light <> 2 THEN
		pc_Shutdown.START := TRUE;
		pc_Shutdown2.START := TRUE;
		SystemPowerButton_Light := 2;
	ELSIF SystemPowerButton_Light = 2 THEN
		pc_AbortShutdown.START := TRUE;
		pc_AbortShutdown2.START := TRUE;
		SystemPowerButton_Light := 1;
	END_IF
END_IF

IF pc_Shutdown.BUSY THEN
	pc_Shutdown.START := FALSE;
END_IF

IF pc_Shutdown2.BUSY THEN
	pc_Shutdown2.START := FALSE;
END_IF

IF pc_AbortShutdown.BUSY THEN
	pc_AbortShutdown.START := FALSE;
END_IF

IF pc_AbortShutdown2.BUSY  THEN
	pc_AbortShutdown2.START := FALSE;
END_IF

pc_Shutdown(
	NETID:= '192.168.31.180.1.1', 
	DELAY:= 10
);

pc_Shutdown2(
	NETID:= '0.0.0.0.1.1', 
	DELAY:= 15
);

pc_AbortShutdown(
	NETID:= '192.168.31.180.1.1', 
);

pc_AbortShutdown2(
	NETID:= '0.0.0.0.1.1'
);
END_ACTION

PROPERTY ResetButton_Light : USINT
GET
ResetButton_Light := _ResetButton_Light;
END_GET
SET
_ResetButton_Light := ResetButton_Light;
END_SET
END_PROPERTY

ACTION ResetButtonAction:
IF SystemError THEN
	ResetButton_Light := 2;
ELSE
	ResetButton_Light := 0;
END_IF

IF ResetButton AND SystemError THEN
	SystemError := FALSE;
END_IF
END_ACTION

PROPERTY StartButton_Light : usint
GET
StartButton_Light := _StartButton_Light;
END_GET
SET
_StartButton_Light := StartButton_Light;
END_SET
END_PROPERTY

ACTION StartButtonAction:
IF AutoMain.step = 0 OR AutoMain.step > 2000 THEN
	Button.StartButton_Light := 0;
END_IF

StartButton_LDP(CLK:=StartButton);
IF StartButton_LDP.q AND LEN(ProjectData.WorkOrder_Now.steel_id) > 0 AND 
	_StartButton_Light = 0 AND NOT AutoMain.bBuzy THEN
	AutoMain.ReStart();
END_IF
END_ACTION

ACTION StepButtonAction:
IF NOT Hmi_Web.Auto_Step_mode_Enable THEN
	Button.StartButton_Light := 0;
ELSE
	IF Hmi_Web.Auto_Step_active THEN
		Button.StartButton_Light := 1;
	ELSE
		Button.StartButton_Light := 2;
	END_IF
END_IF

// StepButton(CLK := StepButton);
IF jogbtn_trig.Q THEN
	IF AutoMain.step > 0 AND AutoMain.step < 2000 THEN
		AutoMain.JogMode();
	ELSIF AutoMain.step = 8001 THEN
		AutoMain.JogMode_Exit();
	END_IF
END_IF
END_ACTION

PROPERTY StepModeButtonLight : usint
GET
StepModeButtonLight := _StepModeButtonLight;
END_GET
SET
_StepModeButtonLight := StepModeButtonLight;
END_SET
END_PROPERTY

PROPERTY StopButton_Light : USINT
GET
StopButton_Light := _StopButton_Light;
END_GET
SET
_StopButton_Light := StopButton_Light;
END_SET
END_PROPERTY

PROPERTY SystemPowerButton_Light : usint
GET
SystemPowerButton_Light := _SystemPowerButton_Light;
END_GET
SET
_SystemPowerButton_Light := SystemPowerButton_Light;
END_SET
END_PROPERTY

END_PROGRAM

// ---- POUs/硬體控制/其他控制/三色燈/LightTower.TcPOU
PROGRAM LightTower
VAR
	tmr1: TON := (PT := TIME#650MS);
	tmr2: TON := (PT := TIME#650MS);
	GreenLight: BOOL;
	YellowLight: BOOL;
	RedLight: BOOL;
	Buzzy: BOOL;
	tmr10: TON;
	halfPass: BOOL;
	tmr1_tmp: BOOL;
	trig: R_TRIG;
	tmr11: TOF;
	tmr5: TON;
	tmr6: TON;
END_VAR

VAR_OUTPUT
	clk : BOOL;
END_VAR

IF tmr1.Q <> tmr1_tmp THEN
	tmr1_tmp := tmr1.Q;
	halfPass := TRUE;
END_IF

IF tmr10.Q THEN
	halfPass:=FALSE;
END_IF

// trig(clk:=door);
// IF trig.Q AND NOT(tmr11.q)THEN
// 	halfPass := TRUE;
// END_IF
// 
// tmr11(in:= door, PT:=T#1S);

CASE hmi.State OF
	// 緊急停止
	MachineState.emergency :
		GreenLight := FALSE;
		YellowLight := FALSE;
		RedLight := tmr1.Q;
		buzzy := FALSE;
		tmr1.PT := T#1S200MS;
		tmr10.PT := T#50MS;
		
	// 安全光柵觸發
	MachineState.Door :
		GreenLight := FALSE;
		YellowLight := NOT(door) AND tmr1.Q;
		RedLight := door AND tmr1.Q;
		buzzy := tmr1.Q AND door;
		tmr1.PT := T#1S200MS;
		tmr10.PT := T#50MS;	
	
	// 發生錯誤
	MachineState.error :
		GreenLight := FALSE;
		YellowLight := FALSE;
		RedLight := tmr1.Q;
		buzzy := tmr1.Q;
	
	// 自動模式
	MachineState.auto_mode :
		GreenLight := tmr1.Q;
		YellowLight := FALSE;
		RedLight := FALSE;
		buzzy := halfPass AND ExpConver.Feed_bBuzy;
		tmr1.PT := T#833MS;
		tmr10.PT := T#50MS;
		
	MachineState.auto_mode_wait :
		GreenLight := tmr1.Q;
		YellowLight := NOT tmr1.Q;
		RedLight := FALSE;
		buzzy := halfPass AND ExpConver.Feed_bBuzy;
		tmr1.PT := T#833MS;
		tmr10.PT := T#50MS;
		
	// 自動模式
// 	MachineState.Remote_Auto_mode :
// 		GreenLight := tmr1.Q;
// 		YellowLight := FALSE;
// 		RedLight := FALSE;
// 		buzzy := halfPass AND ExpConver.Feed_bBuzy;
// 		tmr1.PT := T#650MS;
// 		tmr10.PT := T#50MS;
		
	// 手動模式
	MachineState.manual_mode :
		GreenLight := FALSE;
		YellowLight := tmr1.Q;
		RedLight := FALSE;
		
//		IF axis.AxisMove THEN
//			buzzy := halfPass AND NOT hmi.MainPage_Pause;
//		ELSE
//			buzzy := FALSE;
//		END_IF
		tmr1.PT := T#650MS;
		
	// 歸零模式
	MachineState.Homing_mode :
		GreenLight := tmr1.Q;
		YellowLight := FALSE;
		RedLight := FALSE;
		buzzy := halfPass AND NOT(hmi.Auto_Pause);
		tmr1.PT := T#650MS;
		tmr10.PT := T#100MS;
		
	// 待命
	MachineState.standby :
		GreenLight := TRUE;
		YellowLight := FALSE;
		RedLight := FALSE;
		buzzy := FALSE;
		tmr10.PT := T#50MS;
	
END_CASE

tmr2.PT := tmr1.PT;
tmr1(in:=NOT tmr2.q);
tmr2(in:=tmr1.q);

tmr5(in:=NOT tmr6.q, pt:=T#50MS);
tmr6(in:=tmr5.q, pt:=T#50ms);

tmr10(in:=halfPass);

clk := tmr1.q;

io.q113:= GreenLight;
io.q114:= YellowLight;
io.q115:= RedLight;
io.q116:= buzzy;


// 第2組
// io3.y107:= GreenLight;
// io3.y108:= YellowLight;
// io3.y106:= RedLight;
// io3.Y109:= buzzy;

END_PROGRAM

// ---- POUs/硬體控制/手搖輪/Jog_MPG.TcPOU
PROGRAM Jog_MPG
VAR
	AxisMPG : AXIS_REF;
	
	step: INT;

	
	in_iAxisGroup : dINT;
	
	in_bSpeedSelect1: BOOL;
	in_bSpeedSelect2: BOOL;
	
	in_bAxisSelect1 : BOOL;
	in_bAxisSelect2 : BOOL;
	in_bAxisSelect3 : BOOL;
	
	SpeedSelect: WORD;
	AxisSelect: WORD;
	AxisSelect_old: WORD;
	
	Estop_Trig : R_TRIG;
	
	
(* ============== 軸耦合 功能塊 ==============*)
	AxisGearIn				: MC_GearInDyn;
	AxisMpg_WriteParameter	: MC_WriteParameter;
	AxisMpg_WriteBoolParameter	: MC_WriteBoolParameter;
	AxisReadError			: MC_ReadAxisError;
	AxisReset				: MC_Reset;
	
(* ============== 耦合的軸 ==============*)
	Axis1: POINTER TO AXIS_REF;
	
	i_AxisConrtol : I_Axis;
	
	AxisS			: Sub_Step;
	
	AxisState : ST_AxisStatus;
	
	Speed: LREAL;
	AxisGroup: WORD;
	tmr01: TON;
	
	
	P_Limite: POINTER TO BOOL;
	P_Limite_R_Trig: R_TRIG;
	P_Limite_F_Trig: F_TRIG;
	
	N_Limite: POINTER TO BOOL;
	N_Limite_R_Trig: R_TRIG;
	N_Limite_F_Trig: F_TRIG;
END_VAR

VAR_OUTPUT
	Active  : BOOL;
	// 錯誤步驟
	iErrorID	: INT;
END_VAR

VAR CONSTANT
	// // 軸名稱
	scAxisName: WSTRING := "MPG軸";
END_VAR

_IO();

speed :=  0.01 * EXPT(10,SpeedSelect);
		
AxisGroup := DINT_TO_WORD(in_iAxisGroup * 16#10);

AxisSelect := AxisSelect + AxisGroup;

Active := step > 0 AND step < 10000;

Estop_Trig(CLK:= SystemError);

IF Estop_Trig.Q THEN
	step:=100;
END_IF

IF ProgramReset THEN
	step := 0;
END_IF

AxisMPG.ReadStatus();

IF i_AxisConrtol <> 0 THEN
	AxisState := i_AxisConrtol.Axis_States;
END_IF

_Step0();



AxisGearIn.GearRatio := Speed;



_MC_FB();
tmr01();

ACTION _AxisSet:
CASE AxisSelect OF
// =============== 軸群組A ===============
	16#11:
		i_AxisConrtol := GaX;
		Axis1 := ADR(Axis.Axis_AX);
		
	16#12:
		i_AxisConrtol := GaY;
		Axis1 := ADR(Axis.Axis_AY);
		
	16#13:
		i_AxisConrtol := GaZ;
		Axis1 := ADR(Axis.Axis_AZ1);
		
// =============== 軸群組B ===============
	16#21:
		i_AxisConrtol := GbX;
		Axis1 := ADR(Axis.Axis_BX);
		
	16#22:
		i_AxisConrtol := GbY;
		Axis1 := ADR(Axis.Axis_BY1);
		
	16#23:
		i_AxisConrtol := GbZ;
		Axis1 := ADR(Axis.Axis_BZ);
		
// =============== 軸群組C ===============
	16#31:
		i_AxisConrtol := GcX;
		Axis1 := ADR(Axis.Axis_CX);
		
	16#32:
		i_AxisConrtol := GcY;
		Axis1 := ADR(Axis.Axis_CY);
		
	16#33:
		i_AxisConrtol := GcZ;
		Axis1 := ADR(Axis.Axis_CZ1);
		
// =============== 軸群組D ===============
	16#41:
		i_AxisConrtol := GdX;
		Axis1 := ADR(Axis.Axis_DX);
		
	16#42:
		i_AxisConrtol := GdY;
		Axis1 := ADR(Axis.Axis_DY);
		
	16#43:
		i_AxisConrtol := GdZ;
		Axis1 := ADR(Axis.Axis_DZ);
		
	ELSE
		Axis1 := 0;
		P_Limite := ADR(GaX.OutLimiter);
		N_Limite := ADR(GaX.inLimiter);
END_CASE
END_ACTION

ACTION _IO:
in_bSpeedSelect1 := IO.i604;
in_bSpeedSelect2 := IO.i605;

in_bAxisSelect1 := IO.i601;
in_bAxisSelect2 := IO.i602;
in_bAxisSelect3 := IO.i603;

in_iAxisGroup := Hmi_Web.Jog_GroupSelect;



SpeedSelect.0:= in_bSpeedSelect1;
SpeedSelect.1:= in_bSpeedSelect2;



AxisSelect := 0;
AxisSelect.0 := in_bAxisSelect1;
AxisSelect.1 := in_bAxisSelect2;
AxisSelect.2 := in_bAxisSelect3;
END_ACTION

ACTION _MC_FB:
IF Axis1 > 0 THEN
	AxisGearIn(master := AxisMPG, slave := Axis1^);
END_IF

AxisMpg_WriteParameter(Axis:= AxisMPG);

AxisMpg_WriteBoolParameter(Axis := AxisMPG);

AxisReset(Axis:= AxisMPG);

AxisReadError(Enable:=(step > 0),	Axis := AxisMPG);
END_ACTION

ACTION _Step0:
IF P_Limite > 0 AND N_Limite > 0 THEN
	P_Limite_R_Trig(clk := P_Limite^);
	P_Limite_F_Trig(clk := P_Limite^);
	N_Limite_R_Trig(clk := N_Limite^);
	N_Limite_F_Trig(clk := N_Limite^);
END_IF

CASE step OF
	1:
		AxisReset.Execute := FALSE;
		IF AxisGearIn.Enable OR AxisGearIn.Active THEN
			step := 200;
		ELSE
			step := step + 1;
		END_IF


(* ===================== MPG軸的錯誤重置 ===================== *)
	2:
		IF AxisMPG.Status.Error THEN
			step := step + 1;
		ELSE
			step := 10;
		END_IF
		
	3:
		AxisReset.Execute :=TRUE;
		step := step + 1;
		
	4:
		tmr01.pt := T#500MS;
		tmr01.in := TRUE;
		IF tmr01.q THEN
			tmr01.in := FALSE;
			step := step + 1;
		END_IF
		
	5:
		IF NOT AxisMPG.Status.Error AND AxisReset.Done THEN
			AxisReset.Execute :=FALSE;
			step := 10;
		ELSIF AxisReset.Error THEN
			pMsg.Push_Error(
				ErrorCodeConver.Str(str0:= scAxisName, str1:= ": MPG無法重置", ErrorCode:= AxisReset.ErrorID)
			);
			AxisReset.Execute :=FALSE;
			step:=step + 10000;
		END_IF
		
		
(* ===================== 映射要操作的軸 ===================== *)
	10: // 設定要操作的軸
		_AxisSet();
		step := step + 1;
		
	11:
		tmr01.pt := T#100MS;
		tmr01.in := TRUE;
		IF tmr01.q THEN
			tmr01.in := FALSE;
			step := step + 1;
		END_IF
		
	12: // 確認軸已被設定
		IF i_AxisConrtol <> 0 THEN
			step := step + 1;
		ELSE
			step := 40;
		END_IF
		
	13: // 啟動軸電源
		i_AxisConrtol.PowerOn();
		step := step + 1;
		
	14: // 確認軸啟動狀態
		IF AxisState.Operational THEN
			step := step + 1;
		ELSIF Axis1^.Status.Error THEN
			Hmi.MPG_Mode := FALSE;
			step := 0;
		END_IF
		
	
	15:
		step := 20;
		
		
(* ===================== MPG軸 與 選擇的軸 連接 ===================== *)		
	20:
//		AxisGearIn.Acceleration := 100;
		AxisGearIn.Enable :=TRUE;
		step := step + 1;
		
	21:
		IF AxisGearIn.Active THEN
			step := step + 1;
		END_IF
		
	22:
		step := 30;
		
		
(* ===================== 檢查選擇的軸是否有變更 ===================== *)
	30:
		IF AxisSelect <> AxisSelect_old THEN
		 	step := step + 10;
		ELSIF AxisGearIn.Error THEN
			step := 100;
			pMsg.Push_Error(
				ErrorCodeConver.Str(str0:= scAxisName, str1:= ": GearIn發生錯誤", ErrorCode:= AxisGearIn.ErrorID)
			);
		ELSIF AxisReadError.Valid AND AxisReadError.AxisErrorID > 0 THEN
			IF AxisReadError.AxisErrorID = 16#42A0 THEN
				pMsg.Push_Alarm_NoPause(
					ErrorCodeConver.Str(str0:= scAxisName, str1:= ": 驅動軸到達極限位置", ErrorCode:= AxisReadError.ErrorID)
				);
				step := step + 1;
			ELSIF AxisReadError.AxisErrorID = 16#4462 THEN
				pMsg.Push_Alarm_NoPause(
					ErrorCodeConver.Str(str0:= scAxisName, str1:= ": 驅動軸到負極限開關", ErrorCode:= AxisReadError.ErrorID)
				);
				step := step + 1;
			ELSIF AxisReadError.AxisErrorID = 16#4463 THEN
				pMsg.Push_Alarm_NoPause(
					ErrorCodeConver.Str(str0:= scAxisName, str1:= ": 驅動軸到正極限開關", ErrorCode:= AxisReadError.ErrorID)
				);
				step := step + 1;
			ELSE
				pMsg.Push_Alarm_NoPause(
					ErrorCodeConver.Str(str0:= scAxisName, str1:= ": 軸發生錯誤", ErrorCode:= AxisReadError.ErrorID)
				);
				step := 200;
			END_IF
			
		END_IF
		
	31:
		tmr01.pt := T#1S;
		tmr01.in := TRUE;
		IF tmr01.q THEN
			tmr01.in := FALSE;
			step := 200;
		END_IF
		

(* ===================== 選擇的軸變更 ===================== *)
	40:
		tmr01.pt := T#250MS;
		tmr01.in := TRUE;
		IF tmr01.q THEN
			tmr01.in := FALSE;
			step := step + 1;
		END_IF
		
	41:
		IF AxisSelect <> AxisSelect_old THEN
			AxisSelect_old := AxisSelect;
			step := 200;
		ELSIF Axis1 = 0 THEN
			step := 100;
		ELSE
			step := 30;
		END_IF
			
		
		
		
	
		
	100: // 解耦 檢查參考是否可用
		IF i_AxisConrtol <> 0 THEN
			step := step + 1;
		ELSE
			step := 0;
		END_IF
		
	101:// 停止軸
		IF Axis1 = 0 THEN
			step := 0;
		ELSE
			AxisGearIn.Enable := FALSE;
			step := step + 1;
		END_IF
		
	102:
		i_AxisConrtol.Stop();
		step := step + 1;
		
	103:
		IF AxisS.bBuzy OR AxisS.bError THEN
			step := step + 1;
		END_IF
		
	104:
		IF AxisState.NotMoving THEN
			step := 0;
		ELSE
			step := step + 10000;
		END_IF
		
		
		
		
		
	200: // 切換軸
		IF i_AxisConrtol <> 0 THEN
			step := step + 1;
		ELSE
			step := 0;
		END_IF
	
	201:
		IF Axis1 = 0 THEN
			step := 0;
		ELSE
			AxisGearIn.Enable := FALSE;
			step := step + 1;
		END_IF
		
	202:
		i_AxisConrtol.Stop();
		step := step + 1;
		
	203:
		IF AxisS.bBuzy OR AxisS.bError THEN
			step := step + 1;
		END_IF
		
	204:
		IF AxisState.NotMoving THEN
			step := step + 1;
		ELSIF AxisS.bError THEN
			step := step + 10000;
		END_IF
		
	205:
		Axis1 := 0;
		step := step + 1;
		
	206:
		tmr01.pt := T#150MS;
		tmr01.in := TRUE;
		IF tmr01.q THEN
			tmr01.in := FALSE;
			step := step + 1;
		END_IF
		
	207:
		IF NOT Safety.SystemError AND (AxisSelect MOD 16) <> 0 THEN
			step := 1;
		END_IF
		
	
END_CASE
END_ACTION

METHOD Start : BOOL
VAR_INPUT
END_VAR
step := 1;
END_METHOD

METHOD Stop : BOOL
VAR_INPUT
END_VAR
step := 100;
END_METHOD

END_PROGRAM

// ---- POUs/功能塊/ErrorCodeConver.TcPOU
PROGRAM ErrorCodeConver
VAR
	
END_VAR

METHOD StoberErrorCode : WSTRING
VAR_INPUT
	Name : WSTRING;
	Event : UDINT;
	Cause : UDINT;
END_VAR

VAR
	strtmp1: WSTRING;
	strtmp2: WSTRING;
END_VAR




strtmp2 := WCONCAT(STR1:= Name, STR2:= ":錯誤 Event:");

strtmp1 := UDINT_TO_WSTRING(Event);

strtmp2 := WCONCAT(STR1:= strtmp2, STR2:= strtmp1 );

strtmp2:= WCONCAT(STR1:= strtmp2, STR2:= "Cause:");

strtmp1 := UDINT_TO_WSTRING(Cause);

strtmp2:= WCONCAT(STR1:= strtmp2, STR2:= strtmp1);

// 輸出結果字串

StoberErrorCode := strtmp2;
END_METHOD

METHOD Str : WSTRING
VAR_INPUT
	str0 : WSTRING;
	str1 : WSTRING := "";
	str2 : WSTRING := "";
	str3 : WSTRING := "";
	str4 : WSTRING := "";
	ErrorCode :DWORD;
END_VAR

VAR
	strtmp1: STRING;
	strtmp2: WSTRING;
END_VAR
IF ErrorCode > 16#FFFF THEN
	strtmp1 := DWORD_TO_HEXSTR(in:= ErrorCode, iPrecision:= 8, bLoCase:= FALSE);
ELSE
	strtmp1 := DWORD_TO_HEXSTR(in:= ErrorCode, iPrecision:= 4, bLoCase:= FALSE);
END_IF

strtmp2 := STRING_TO_WSTRING(strtmp1);

strtmp2 := WCONCAT(STR1:= "(0x", STR2:= strtmp2);

strtmp2 := WCONCAT(STR1:= strtmp2, STR2:= ")" );

strtmp2:= WCONCAT(STR1:= str4, STR2:= strtmp2);

strtmp2:= WCONCAT(STR1:= str3, STR2:= strtmp2);

strtmp2:= WCONCAT(STR1:= str2, STR2:= strtmp2);

strtmp2:= WCONCAT(STR1:= str1, STR2:= strtmp2);

Str:= WCONCAT(STR1:= str0, STR2:= strtmp2);
END_METHOD

END_PROGRAM

// ---- POUs/功能塊/EtherCat相關/GetEtherSta.TcPOU
PROGRAM GetEtherSta
VAR
	fbGetAllSlaveStates : FB_EcGetAllSlaveStates;
    sNetId1      AT %I*  : AMSNETID ;
	sNetId2      AT %I*  : AMSNETID ;
    bExecute            : BOOL;
	
    devStates1				: ARRAY[0..255] OF ST_EcSlaveState;
	devStates2				: ARRAY[0..255] OF ST_EcSlaveState;
	devStates1_old			: ARRAY[0..255] OF BYTE;
	devStates2_old			: ARRAY[0..255] OF BYTE;
	Ethercat_1_IsAlarm		: BOOL;
	Ethercat_2_IsAlarm		: BOOL;
	
    nSlaves             : UINT := 0;
	nSlaves2             : UINT := 0;
    nErrId              : UDINT;
	
	fbEcReqSlaveState : FB_EcReqSlaveState;
	
	fb_EcGetSlaveTopologyInfo	: FB_EcGetConfSlaves;
	SlaveData1 				: ARRAY[0..255] OF ST_EcSlaveConfigData;
	SlaveData2 				: ARRAY[0..255] OF ST_EcSlaveConfigData;
	
	step: INT;
	tmr1: TON;
	i: UINT;
	
	fb_EcSetSlaveState : FB_EcSetSlaveState;
	resetSlaveNumber : INT;
	tmr100: TON;
	str_TmpString: WSTRING;
	
	
	
	step100: INT;
END_VAR

VAR_OUTPUT
	bErrorGetEC: BOOL;

	bBuzy: BOOL;
	bError: BOOL;
	bDone: BOOL;
	iErrorId : INT;
END_VAR

fbGetAllSlaveStates();
bErrorGetEC := fbGetAllSlaveStates.bError;
nErrId := fbGetAllSlaveStates.nErrId;

CASE step OF
	0:
		fb_EcGetSlaveTopologyInfo.sNetId	:= F_CreateAmsNetId(sNetId1);
		fb_EcGetSlaveTopologyInfo.pArrEcConfSlaveInfo	:= ADR(SlaveData1);
		fb_EcGetSlaveTopologyInfo.cbBufLen	:= SIZEOF(SlaveData1);
		fb_EcGetSlaveTopologyInfo.bExecute	:= TRUE;
		step := step + 1;
		
	1:
		IF fb_EcGetSlaveTopologyInfo.bBusy OR fb_EcGetSlaveTopologyInfo.bError THEN
			step := step + 1;
		END_IF
		
	2:
		IF NOT fb_EcGetSlaveTopologyInfo.bBusy THEN
			fb_EcGetSlaveTopologyInfo.bExecute := FALSE;
			step := step + 1;
		END_IF
		
	3:
		fb_EcGetSlaveTopologyInfo.sNetId	:= F_CreateAmsNetId(sNetId2);
		fb_EcGetSlaveTopologyInfo.pArrEcConfSlaveInfo	:= ADR(SlaveData2);
		fb_EcGetSlaveTopologyInfo.cbBufLen	:= SIZEOF(SlaveData2);
		fb_EcGetSlaveTopologyInfo.bExecute	:= TRUE;
		step := step + 1;
		
	4:
		IF fb_EcGetSlaveTopologyInfo.bBusy OR fb_EcGetSlaveTopologyInfo.bError THEN
			step := step + 1;
		END_IF
		
	5:
		IF NOT fb_EcGetSlaveTopologyInfo.bBusy THEN
			fb_EcGetSlaveTopologyInfo.bExecute := FALSE;
			step := step + 1;
		END_IF
		
	6:
		tmr1.in := TRUE;
		tmr1.pt := T#10S;
		IF tmr1.Q THEN
			tmr1.in := FALSE;
			step := step + 1;
		END_IF
		step := 10;
		
		
	10:
		fbGetAllSlaveStates.sNetId:= F_CreateAmsNetId(sNetId1);
		fbGetAllSlaveStates.pStateBuf	:= ADR(devStates1);
		fbGetAllSlaveStates.cbBufLen	:= SIZEOF(devStates1);
		fbGetAllSlaveStates.bExecute := TRUE;
		step := step + 1;
		
	11:
		IF fbGetAllSlaveStates.bBusy OR fbGetAllSlaveStates.bError THEN
			step := step + 1;
		END_IF
		
	12:
		IF NOT fbGetAllSlaveStates.bBusy THEN
			fbGetAllSlaveStates.bExecute := FALSE;
			nSlaves := fbGetAllSlaveStates.nSlaves;
			step := step + 1;
		END_IF
		
	13:
		fbGetAllSlaveStates.sNetId		:= F_CreateAmsNetId(sNetId2);
		fbGetAllSlaveStates.pStateBuf	:= ADR(devStates2);
		fbGetAllSlaveStates.cbBufLen	:= SIZEOF(devStates2);
		fbGetAllSlaveStates.bExecute := TRUE;
		step := step + 1;
		
	14:
		IF fbGetAllSlaveStates.bBusy OR fbGetAllSlaveStates.bError THEN
			step := step + 1;
		END_IF
		
	15:
		IF NOT fbGetAllSlaveStates.bBusy THEN
			fbGetAllSlaveStates.bExecute := FALSE;
			nSlaves2 := fbGetAllSlaveStates.nSlaves;
			step := step + 1;
		END_IF
		
	16:
		FOR i := 0 TO nSlaves - 1 DO
			IF devStates1[i].deviceState <> devStates1_old[i] THEN
				IF NOT Ethercat_1_IsAlarm AND (devStates1[i].deviceState AND 16#F) <> 8 THEN
					pMsg.Push_Alarm_NoPause("EtherCat網路1裝置:", TO_WSTRING(SlaveData1[i].sName), "狀態為", EtherCAT_Status(devStates1[i].deviceState));
					Ethercat_1_IsAlarm := TRUE;
				END_IF
				devStates1_old[i] := devStates1[i].deviceState;
			END_IF
		END_FOR
		
		FOR i := 0 TO nSlaves2 - 1 DO
			IF devStates2[i].deviceState <> devStates2_old[i] THEN
				IF NOT Ethercat_2_IsAlarm AND (devStates2[i].deviceState AND 16#F) <> 8 THEN
					pMsg.Push_Alarm_NoPause("EtherCat網路1裝置:", TO_WSTRING(SlaveData2[i].sName), "狀態為", EtherCAT_Status(devStates2[i].deviceState));
					Ethercat_2_IsAlarm := TRUE;
				END_IF
				devStates2_old[i] := devStates2[i].deviceState;
			END_IF
		END_FOR
		step := step + 1;
		
		
	17:
		Ethercat_1_IsAlarm := FALSE;
		Ethercat_2_IsAlarm := FALSE;
		step := 20;
		
	20:
		
		tmr1.in := TRUE;
		tmr1.pt := T#5S;
		IF tmr1.Q THEN
			tmr1.in := FALSE;
			step := step + 1;
		END_IF
		
	21:
		step := 10;
			
		
END_CASE

fb_EcGetSlaveTopologyInfo();

fbEcReqSlaveState();

Step100_resetECAT();

tmr1();

METHOD ResetECat1 : BOOL
VAR_INPUT
	SlaveAddr : INT;
	
END_VAR
resetSlaveNumber := SlaveAddr;
fb_EcSetSlaveState.sNetId := F_CreateAmsNetId(sNetId1);
bDone := FALSE;
step100 := 100;
END_METHOD

METHOD ResetECat2 : BOOL
VAR_INPUT
	SlaveAddr : INT;
	
END_VAR
resetSlaveNumber := SlaveAddr;
fb_EcSetSlaveState.sNetId := F_CreateAmsNetId(sNetId2);
bDone := FALSE;
step100 := 100;
END_METHOD

ACTION Step100_resetECAT:
bBuzy := step100 > 0 AND step100 < 10000;
bError := step100 > 10000;

IF (EStop OR SystemError) THEN
	bDone := FALSE;
	IF bBuzy THEN
		step100 := step100  + 10000;
	END_IF
END_IF

IF ProgramReset THEN
	iErrorId := step;
	step := 0;
END_IF

CASE step100 OF
	100:
		fb_EcSetSlaveState.bExecute := FALSE;
		fb_EcSetSlaveState.tTimeout := T#5S;
		step100 := step100 + 1;
		
	101:// 將裝置設定狀態設為init
		fb_EcSetSlaveState.nSlaveAddr := INT_TO_UINT(resetSlaveNumber);
		fb_EcSetSlaveState.reqState := 1;
		fb_EcSetSlaveState.bExecute := TRUE;
		step100 := step100 + 1;
		
		
	102:
		IF fb_EcSetSlaveState.bBusy OR fb_EcSetSlaveState.bError THEN
			step100 := step100 + 1;
		END_IF
		
	103:
		IF fb_EcSetSlaveState.currState.deviceState = 1 THEN
			fb_EcSetSlaveState.bExecute := FALSE;
			step100 := step100 + 1;
		ELSIF fb_EcSetSlaveState.bError THEN
			fb_EcSetSlaveState.bExecute := FALSE;
			str_TmpString := WCONCAT(STR1:= "設定EtherCat站號", STR2:= INT_TO_WSTRING(resetSlaveNumber));
			str_TmpString := WCONCAT(STR1:= str_TmpString, STR2:= " 的狀態為INIT時發生錯誤");
			pMsg.Push_Alarm(str_TmpString);
			step100 := step100 + 10000;
		END_IF
	
	104:
		tmr100.IN:=TRUE;
		tmr100.PT := T#500MS;
		IF tmr100.Q THEN
			tmr100.IN:=FALSE;
			step100 := step100 + 1;
		END_IF
		
	105:
		step100 := 110;
		
		
		
	110:// 將裝置設定狀態設為PREOP 
		fb_EcSetSlaveState.nSlaveAddr := INT_TO_UINT(resetSlaveNumber);
		fb_EcSetSlaveState.reqState := 2;
		fb_EcSetSlaveState.bExecute := TRUE;
		step100 := step100 + 1;
		
	111:
		IF fb_EcSetSlaveState.bBusy OR fb_EcSetSlaveState.bError THEN
			step100 := step100 + 1;
		END_IF
		
	112:
		IF fb_EcSetSlaveState.currState.deviceState = 2 THEN
			fb_EcSetSlaveState.bExecute := FALSE;
			step100 := step100 + 1;
		ELSIF fb_EcSetSlaveState.bError THEN
			fb_EcSetSlaveState.bExecute := FALSE;
			str_TmpString := WCONCAT(STR1:= "設定EtherCat站號", STR2:= INT_TO_WSTRING(resetSlaveNumber));
			str_TmpString := WCONCAT(STR1:= str_TmpString, STR2:= " 的狀態為PREOP時發生錯誤");
			pMsg.Push_Alarm(str_TmpString);
			step100 := step100 + 10000;
		END_IF
		
	113:
		tmr100.IN:=TRUE;
		tmr100.PT := T#500MS;
		IF tmr100.Q THEN
			tmr100.IN:=FALSE;
			step100 := step100 + 1;
		END_IF
		
	114:
		step100 := 120;
		
		
		
	120:// 將裝置設定狀態設為SAFEOP
		fb_EcSetSlaveState.nSlaveAddr := INT_TO_UINT(resetSlaveNumber);
		fb_EcSetSlaveState.reqState := 4;
		fb_EcSetSlaveState.bExecute := TRUE;
		step100 := step100 + 1;
		
		
	121:
		IF fb_EcSetSlaveState.bBusy OR fb_EcSetSlaveState.bError THEN
			step100 := step100 + 1;
		END_IF
		
	122:
		IF fb_EcSetSlaveState.currState.deviceState = 4 THEN
			fb_EcSetSlaveState.bExecute := FALSE;
			step100 := step100 + 1;
		ELSIF fb_EcSetSlaveState.bError THEN
			fb_EcSetSlaveState.bExecute := FALSE;
			str_TmpString := WCONCAT(STR1:= "設定EtherCat站號", STR2:= INT_TO_WSTRING(resetSlaveNumber));
			str_TmpString := WCONCAT(STR1:= str_TmpString, STR2:= " 的狀態為SAFEOP時發生錯誤");
			pMsg.Push_Alarm(str_TmpString);
			step100 := step100 + 10000;
		END_IF
		
	123:
		tmr100.IN:=TRUE;
		tmr100.PT := T#500MS;
		IF tmr100.Q THEN
			tmr100.IN:=FALSE;
			step100 := step100 + 1;
		END_IF
		
	124:
		step100 := 130;
		
	130:// 將裝置設定狀態設為OP
		fb_EcSetSlaveState.nSlaveAddr := INT_TO_UINT(resetSlaveNumber);
		fb_EcSetSlaveState.reqState := 8;
		fb_EcSetSlaveState.bExecute := TRUE;
		step100 := step100 + 1;
		
		
	131:
		IF fb_EcSetSlaveState.bBusy OR fb_EcSetSlaveState.bError THEN
			step100 := step100 + 1;
		END_IF
		
	132:
		IF fb_EcSetSlaveState.currState.deviceState = 8 THEN
			fb_EcSetSlaveState.bExecute := FALSE;
			step100 := step100 + 1;
		ELSIF fb_EcSetSlaveState.bError THEN
			fb_EcSetSlaveState.bExecute := FALSE;
			str_TmpString := WCONCAT(STR1:= "設定EtherCat站號", STR2:= INT_TO_WSTRING(resetSlaveNumber));
			str_TmpString := WCONCAT(STR1:= str_TmpString, STR2:= " 的狀態為SAFEOP時發生錯誤");
			pMsg.Push_Alarm(str_TmpString);
			step100 := step100 + 10000;
		END_IF
		
	133:
		tmr100.IN:=TRUE;
		tmr100.PT := T#500MS;
		IF tmr100.Q THEN
			tmr100.IN:=FALSE;
			step100 := step100 + 1;
		END_IF
		
	134:
		bDone := TRUE;
		step100 := 0;
		
END_CASE

tmr100();
fb_EcSetSlaveState();
END_ACTION

END_PROGRAM

// ---- POUs/功能塊/EtherCat相關/EtherCAT_Status.TcPOU
FUNCTION EtherCAT_Status : WSTRING
VAR_INPUT
	Status_input : BYTE;
END_VAR
VAR
	Status1 : BYTE;
	Status2 : BYTE;
	OutTmp : WSTRING;
END_VAR

Status1 := (Status_input AND 16#F);
Status2 := (Status_input AND 16#F0);

CASE Status1 OF
	1:
		OutTmp := "INIT";
		
	2:
		OutTmp := "PREOP";
		
	3:
		OutTmp := "BOOTSTRAP";
		
	4:
		OutTmp := "SAFEOP";
		
	8:
		OutTmp := "OP";
END_CASE

OutTmp := WCONCAT(STR1:= OutTmp, STR2:= ",");

CASE Status2 OF
	16#10:
		OutTmp := WCONCAT(STR1:= OutTmp, STR2:= "狀態機錯誤");
		
	16#20:
		OutTmp := WCONCAT(STR1:= OutTmp, STR2:= "無效的產品代碼");
		
	16#40:
		OutTmp := WCONCAT(STR1:= OutTmp, STR2:= "初始化發生錯誤");
		
	16#80:
		OutTmp := WCONCAT(STR1:= OutTmp, STR2:= "從站已停用");
END_CASE

EtherCAT_Status := OutTmp;

END_FUNCTION

// ---- POUs/硬體控制/軸/AxisAction.TcPOU
PROGRAM AxisAction
VAR
	bBoot : BOOL := true;

	bMove: BOOL;
	tof_PowerOff: TOF;
	ldf_PowerOff: F_TRIG;
END_VAR

IF bBoot THEN
	initAction();
	IF GaX.b_ISVALIDREF AND GaY.b_ISVALIDREF AND GaZ.b_ISVALIDREF AND
		GbX.b_ISVALIDREF AND GbY.b_ISVALIDREF AND GbZ.b_ISVALIDREF AND
		GcX.b_ISVALIDREF AND GcY.b_ISVALIDREF AND GcZ.b_ISVALIDREF AND
		GdX.b_ISVALIDREF AND GdY.b_ISVALIDREF AND GdZ.b_ISVALIDREF AND
		Fx.b_ISVALIDREF THEN
			bBoot := FALSE;
	END_IF
END_IF


//
IF MaCfg.bInSite_Invert THEN
	GaX(outLimiter := IO.i303, inLimiter := IO.i304, origin := FALSE);
	GaY(outLimiter := IO.i305, inLimiter := IO.i306, origin := FALSE);
	
	GbX(outLimiter := IO.i403, inLimiter := IO.i404, origin := FALSE);
	GbY(outLimiter := IO.i408, inLimiter := IO.i407, origin := FALSE);

	GcX(outLimiter := IO.i411, inLimiter := IO.i412, origin := FALSE);
	GcY(outLimiter := IO.i413, inLimiter := IO.i414, origin := FALSE);

	GdX(outLimiter := IO.i311, inLimiter := IO.i312, origin := FALSE);
	GdY(outLimiter := IO.i314, inLimiter := IO.i313, origin := FALSE);

ELSE
	GaX(outLimiter := IO.i304, inLimiter := IO.i303, origin := FALSE);
	GaY(outLimiter := IO.i306, inLimiter := IO.i305, origin := FALSE);
	
	GbX(outLimiter := IO.i404, inLimiter := IO.i403, origin := FALSE);
	GbY(outLimiter := IO.i407, inLimiter := IO.i408, origin := FALSE);
	
	GcX(outLimiter := IO.i412, inLimiter := IO.i411, origin := FALSE);
	GcY(outLimiter := IO.i414, inLimiter := IO.i413, origin := FALSE);
	
	GdX(outLimiter := IO.i312, inLimiter := IO.i311, origin := FALSE);
	GdY(outLimiter := IO.i313, inLimiter := IO.i314, origin := FALSE);
END_IF


GaZ(outLimiter := IO.i307, inLimiter := IO.i308 AND IO.i407, origin := FALSE);

GbZ(outLimiter := IO.i406, inLimiter := IO.i405, origin := FALSE);

GcZ(outLimiter := IO.i415, inLimiter := IO.i408, origin := FALSE);

GdZ(outLimiter := IO.i315, inLimiter := IO.i316, origin := FALSE);

Fx(outLimiter := TRUE, inLimiter := TRUE, origin := FALSE);

Jog_MPG();

bIsHome := TRUE;
			
bPower :=	GaX.Axis1Power.Status;
			
bMove := Axis.Axis_AX.Status.Moving;
			
tof_PowerOff(IN:=bMove, PT:=T#30M);
ldf_PowerOff(CLK:=tof_PowerOff.Q);

IF ldf_PowerOff.Q THEN
	GaX.PowerOff();
END_IF

EtherCat_Driver_Reset();

IF HMI.Set_Axis_Limit THEN
	GaX.SetLimit();
	GaY.SetLimit();
	GaZ.SetLimit();
	
	GbX.SetLimit();
	GbZ.SetLimit();
	GbY.SetLimit();
	
	GcX.SetLimit();
	GcY.SetLimit();
	GcZ.SetLimit();
	
	GdX.SetLimit();
	GdY.SetLimit();
	GdZ.SetLimit();
	
	HMI.Set_Axis_Limit := FALSE;
END_IF

ReadStoberError();

Hmi_Web.Jog_Ga.Pos.X := GaX.fPos;
Hmi_Web.Jog_Ga.Pos.Y := GaY.fPos;
Hmi_Web.Jog_Ga.Pos.Z := GaZ.fPos;

Hmi_Web.Jog_Gb.Pos.X := GbX.fPos;
Hmi_Web.Jog_Gb.Pos.Y := GbY.fPos;
Hmi_Web.Jog_Gb.Pos.Z := GbZ.fPos;

Hmi_Web.Jog_Gc.Pos.X := GcX.fPos;
Hmi_Web.Jog_Gc.Pos.Y := GcY.fPos;
Hmi_Web.Jog_Gc.Pos.Z := GcZ.fPos;

Hmi_Web.Jog_Gd.Pos.X := GdX.fPos;
Hmi_Web.Jog_Gd.Pos.Y := GdY.fPos;
Hmi_Web.Jog_Gd.Pos.Z := GdZ.fPos;

METHOD initAction : BOOL
VAR_INPUT
END_VAR
GaX.Axis1 REF= Axis_AX;
GaY.Axis1 REF= Axis_AY;
GaZ.Axis1 REF= Axis_AZ1;
GaZ.Axis2 REF= Axis_AZ2;

GbX.Axis1 REF= Axis_BX;
GbY.Axis1 REF= Axis_BY1;
GbY.Axis2 REF= Axis_BY2;
GbZ.Axis1 REF= Axis_BZ;

GcX.Axis1 REF= Axis_CX;
GcY.Axis1 REF= Axis_CY;
GcZ.Axis1 REF= Axis_CZ1;
GcZ.Axis2 REF= Axis_CZ2;

GdX.Axis1 REF= Axis_DX;
GdY.Axis1 REF= Axis_DY;
GdZ.Axis1 REF= Axis_DZ;

Fx.Axis1 REF= Axis_FX1;
Fx.Axis2 REF= Axis_FX2;

GaX.Name	:= "GaX";
GaY.Name	:= "GaY";
GaZ.Name	:= "GaZ1";
GaZ.Name2	:= "GaZ2";

GbX.Name	:= "GbX";
GbY.Name	:= "GbY1";
GbY.Name2	:= "GbY2";
GbZ.Name	:= "GbZ";

GcX.Name	:= "GcX";
GcY.Name	:= "GcY";
GcZ.Name	:= "GcZ1";
GcZ.Name2	:= "GcZ2";

GdX.Name	:= "GdX";
GdY.Name	:= "GdY";
GdZ.Name	:= "GdZ";

Fx.Name := "Fx1";
Fx.Name2 := "Fx2";

GaX.Set_Recoder(ADR(Axis.GaX_total_Move));
GaY.Set_Recoder(ADR(Axis.GaY_total_Move));
GaZ.Set_Recoder(ADR(Axis.GaZ_total_Move));

GbX.Set_Recoder(ADR(Axis.GbX_total_Move));
GbY.Set_Recoder(ADR(Axis.GbY_total_Move));
GbZ.Set_Recoder(ADR(Axis.GbZ_total_Move));

GcX.Set_Recoder(ADR(Axis.GcX_total_Move));
GcY.Set_Recoder(ADR(Axis.GcY_total_Move));
GcZ.Set_Recoder(ADR(Axis.GcZ_total_Move));

GdX.Set_Recoder(ADR(Axis.GdX_total_Move));
GdY.Set_Recoder(ADR(Axis.GdY_total_Move));
GdZ.Set_Recoder(ADR(Axis.GdZ_total_Move));
END_METHOD

END_PROGRAM

// ---- POUs/功能塊/EtherCat相關/EtherCat_Driver_Reset.TcPOU
PROGRAM EtherCat_Driver_Reset
VAR
	step: INT;
END_VAR

VAR_OUTPUT
	bBuzy: BOOL;
	bError: BOOL;
	bDone: BOOL;
	iErrorId : INT;
END_VAR

bBuzy := step > 0 AND step < 10000;
bError := step >= 10000;

// 緊急狀態
IF (EStop OR SystemError) THEN
	bDone := FALSE;
	IF bBuzy THEN
		step := step  + 10000;
	END_IF
END_IF

IF ProgramReset THEN
	iErrorId := step;
	step := 0;
END_IF

CASE step OF
	1:
		bDone := FALSE;
		step := step + 1;
		
	2:
		step := 10;
		
	10:
		IF GetEtherSta.devStates1[0].deviceState = 8 THEN
			step := step + 10;
		ELSE
			step := step + 1;
		END_IF
		
	11:
		GetEtherSta.ResetECat1(1001);
		step := step + 1;
		
	12:
		IF GetEtherSta.bBuzy OR GetEtherSta.bError THEN
			step := step + 1;
		END_IF
		
	13:
		IF GetEtherSta.bDone THEN
			step := step + 1;
		ELSIF GetEtherSta.bError THEN
			pMsg.Push_Alarm("重置Driver1-1 EtherCat狀態失敗");
			step := step + 10000;
		END_IF
		
	14:
		step := 20;
		
	20:
		IF GetEtherSta.devStates1[1].deviceState = 8 THEN
			step := step + 10;
		ELSE
			step := step + 1;
		END_IF
		
	21:
		GetEtherSta.ResetECat1(1002);
		step := step + 1;
		
	22:
		IF GetEtherSta.bBuzy OR GetEtherSta.bError THEN
			step := step + 1;
		END_IF
		
	23:
		IF GetEtherSta.bDone THEN
			step := step + 1;
		ELSIF GetEtherSta.bError THEN
			pMsg.Push_Alarm("重置Driver1-2 EtherCat狀態失敗");
			step := step + 10000;
		END_IF
		
	24:
		step := 30;
		
	30:
		IF GetEtherSta.devStates1[2].deviceState = 8 THEN
			step := step + 10;
		ELSE
			step := step + 1;
		END_IF
		
	31:
		GetEtherSta.ResetECat1(1002);
		step := step + 1;
		
	32:
		IF GetEtherSta.bBuzy OR GetEtherSta.bError THEN
			step := step + 1;
		END_IF
		
	33:
		IF GetEtherSta.bDone THEN
			step := step + 1;
		ELSIF GetEtherSta.bError THEN
			pMsg.Push_Alarm("重置Driver1-3 EtherCat狀態失敗");
			step := step + 10000;
		END_IF
		
	34:
		step := 40;
		
	40:
		IF GetEtherSta.devStates1[3].deviceState = 8 THEN
			step := step + 10;
		ELSE
			step := step + 1;
		END_IF
		
	41:
		GetEtherSta.ResetECat1(1004);
		step := step + 1;
		
	42:
		IF GetEtherSta.bBuzy OR GetEtherSta.bError THEN
			step := step + 1;
		END_IF
		
	43:
		IF GetEtherSta.bDone THEN
			step := step + 1;
		ELSIF GetEtherSta.bError THEN
			pMsg.Push_Alarm("重置Driver1-4 EtherCat狀態失敗");
			step := step + 10000;
		END_IF
		
	44:
		step := 50;
		
	50:
		step := 100;
		
// 塔電櫃驅動器
	100:
		IF GetEtherSta.devStates2[5].deviceState = 8 THEN
			step := step + 10;
		ELSE
			step := step + 1;
		END_IF
		
	101:
		GetEtherSta.ResetECat2(1006);
		step := step + 1;
		
	102:
		IF GetEtherSta.bBuzy OR GetEtherSta.bError THEN
			step := step + 1;
		END_IF
		
	103:
		IF GetEtherSta.bDone THEN
			step := step + 1;
		ELSIF GetEtherSta.bError THEN
			pMsg.Push_Alarm("重置Driver2-1 EtherCat狀態失敗");
			step := step + 10000;
		END_IF
		
	104:
		step := 110;
		
	110:
		IF GetEtherSta.devStates2[6].deviceState = 8 THEN
			step := step + 10;
		ELSE
			step := step + 1;
		END_IF
		
	111:
		GetEtherSta.ResetECat2(1007);
		step := step + 1;
		
	112:
		IF GetEtherSta.bBuzy OR GetEtherSta.bError THEN
			step := step + 1;
		END_IF
		
	113:
		IF GetEtherSta.bDone THEN
			step := step + 1;
		ELSIF GetEtherSta.bError THEN
			pMsg.Push_Alarm("重置Driver2-2 EtherCat狀態失敗");
			step := step + 10000;
		END_IF
		
	114:
		step := 120;
	// CarRailln	
	120:
		IF GetEtherSta.devStates2[7].deviceState = 8 THEN
			step := step + 10;
		ELSE
			step := step + 1;
		END_IF
		
	121:
		GetEtherSta.ResetECat2(1008);
		step := step + 1;
		
	122:
		IF GetEtherSta.bBuzy OR GetEtherSta.bError THEN
			step := step + 1;
		END_IF
		
	123:
		IF GetEtherSta.bDone THEN
			step := step + 1;
		ELSIF GetEtherSta.bError THEN
			pMsg.Push_Alarm("重置Driver2-3 EtherCat狀態失敗");
			step := step + 10000;
		END_IF
		
	124:
		step := 130;
		
	130:
		IF GetEtherSta.devStates2[8].deviceState = 8 THEN
			step := step + 10;
		ELSE
			step := step + 1;
		END_IF
		
	131:
		GetEtherSta.ResetECat2(1009);
		step := step + 1;
		
	132:
		IF GetEtherSta.bBuzy OR GetEtherSta.bError THEN
			step := step + 1;
		END_IF
		
	133:
		IF GetEtherSta.bDone THEN
			step := step + 1;
		ELSIF GetEtherSta.bError THEN
			pMsg.Push_Alarm("重置Driver2-4 EtherCat狀態失敗");
			step := step + 10000;
		END_IF
		
	134:
		step := 140;
	
	140:
		IF GetEtherSta.devStates2[9].deviceState = 8 THEN
			step := step + 10;
		ELSE
			step := step + 1;
		END_IF
		
	141:
		GetEtherSta.ResetECat2(1010);
		step := step + 1;
		
	142:
		IF GetEtherSta.bBuzy OR GetEtherSta.bError THEN
			step := step + 1;
		END_IF
		
	143:
		IF GetEtherSta.bDone THEN
			step := step + 1;
		ELSIF GetEtherSta.bError THEN
			pMsg.Push_Alarm("重置Driver2-5 EtherCat狀態失敗");
			step := step + 10000;
		END_IF
		
	144:
		step := 150;
		
	150:
		IF GetEtherSta.devStates2[10].deviceState = 8 THEN
			step := step + 10;
		ELSE
			step := step + 1;
		END_IF
		
	151:
		GetEtherSta.ResetECat2(1011);
		step := step + 1;
		
	152:
		IF GetEtherSta.bBuzy OR GetEtherSta.bError THEN
			step := step + 1;
		END_IF
		
	153:
		IF GetEtherSta.bDone THEN
			step := step + 1;
		ELSIF GetEtherSta.bError THEN
			pMsg.Push_Alarm("重置Driver2-6 EtherCat狀態失敗");
			step := step + 10000;
		END_IF
		
	154:
		bDone := TRUE;
		step := 0;
END_CASE

